LIN {X 52, Y 256, Z 47} c_vel
LIN {X 42, Y 261, Z 47} c_vel
LIN {X 30, Y 267, Z 47} c_vel
LIN {X 16, Y 273, Z 47} c_vel
LIN {X 0, Y 278, Z 47} c_vel
LIN {X 14, Y 327, Z 47} c_vel
LIN {X 28, Y 322, Z 47} c_vel
LIN {X 43, Y 317, Z 47} c_vel
LIN {X 57, Y 311, Z 47} c_vel
LIN {X 70, Y 304, Z 47} c_vel
LIN {X 81, Y 298, Z 47} c_vel
LIN {X 90, Y 291, Z 47} c_vel
LIN {X 99, Y 284, Z 47} c_vel
LIN {X 106, Y 277, Z 47} c_vel
LIN {X 113, Y 269, Z 47} c_vel
LIN {X 118, Y 261, Z 47} c_vel
LIN {X 123, Y 253, Z 47} c_vel
LIN {X 127, Y 244, Z 47} c_vel
LIN {X 130, Y 235, Z 47} c_vel
LIN {X 131, Y 226, Z 47} c_vel
LIN {X 133, Y 217, Z 47} c_vel
LIN {X 133, Y 207, Z 47} c_vel
LIN {X 133, Y 197, Z 47} c_vel
LIN {X 131, Y 186, Z 47} c_vel
LIN {X 129, Y 173, Z 47} c_vel
LIN {X 126, Y 160, Z 47} c_vel
LIN {X 120, Y 138, Z 47} c_vel
LIN {X 115, Y 118, Z 47} c_vel
LIN {X 112, Y 106, Z 47} c_vel
LIN {X 111, Y 96, Z 47} c_vel
LIN {X 110, Y 88, Z 47} c_vel
LIN {X 110, Y 81, Z 47} c_vel
LIN {X 111, Y 74, Z 47} c_vel
LIN {X 113, Y 69, Z 47} c_vel
LIN {X 116, Y 63, Z 47} c_vel
LIN {X 119, Y 58, Z 47} c_vel
LIN {X 124, Y 53, Z 47} c_vel
LIN {X 130, Y 48, Z 47} c_vel
LIN {X 138, Y 43, Z 47} c_vel
LIN {X 111, Y 0, Z 47} c_vel
$OUT[4] = FALSE
WAIT SEC 10.0
LIN {X 111, Y 0, Z 48} c_vel
$OUT[4] = TRUE
LIN {X 111, Y 0, Z 48} c_vel
LIN {X 106, Y 3, Z 48} c_vel
LIN {X 97, Y 9, Z 48} c_vel
LIN {X 89, Y 16, Z 48} c_vel
LIN {X 83, Y 23, Z 48} c_vel
LIN {X 77, Y 31, Z 48} c_vel
LIN {X 71, Y 39, Z 48} c_vel
LIN {X 67, Y 47, Z 48} c_vel
LIN {X 64, Y 56, Z 48} c_vel
LIN {X 62, Y 64, Z 48} c_vel
LIN {X 60, Y 73, Z 48} c_vel
LIN {X 59, Y 82, Z 48} c_vel
LIN {X 59, Y 92, Z 48} c_vel
LIN {X 60, Y 103, Z 48} c_vel
LIN {X 62, Y 114, Z 48} c_vel
LIN {X 65, Y 127, Z 48} c_vel
LIN {X 69, Y 144, Z 48} c_vel
LIN {X 74, Y 163, Z 48} c_vel
LIN {X 79, Y 180, Z 48} c_vel
LIN {X 81, Y 191, Z 48} c_vel
LIN {X 82, Y 201, Z 48} c_vel
LIN {X 82, Y 209, Z 48} c_vel
LIN {X 82, Y 217, Z 48} c_vel
LIN {X 80, Y 223, Z 48} c_vel
LIN {X 78, Y 229, Z 48} c_vel
LIN {X 75, Y 234, Z 48} c_vel
LIN {X 71, Y 240, Z 48} c_vel
LIN {X 66, Y 245, Z 48} c_vel
LIN {X 60, Y 250, Z 48} c_vel
LIN {X 52, Y 256, Z 48} c_vel
LIN {X 42, Y 261, Z 48} c_vel
LIN {X 30, Y 267, Z 48} c_vel
LIN {X 16, Y 273, Z 48} c_vel
LIN {X 0, Y 278, Z 48} c_vel
LIN {X 14, Y 327, Z 48} c_vel
LIN {X 28, Y 322, Z 48} c_vel
LIN {X 43, Y 317, Z 48} c_vel
LIN {X 57, Y 311, Z 48} c_vel
LIN {X 70, Y 304, Z 48} c_vel
LIN {X 81, Y 298, Z 48} c_vel
LIN {X 90, Y 291, Z 48} c_vel
LIN {X 99, Y 284, Z 48} c_vel
LIN {X 106, Y 277, Z 48} c_vel
LIN {X 113, Y 269, Z 48} c_vel
LIN {X 118, Y 261, Z 48} c_vel
LIN {X 123, Y 253, Z 48} c_vel
LIN {X 127, Y 244, Z 48} c_vel
LIN {X 130, Y 235, Z 48} c_vel
LIN {X 131, Y 226, Z 48} c_vel
LIN {X 133, Y 217, Z 48} c_vel
LIN {X 133, Y 207, Z 48} c_vel
LIN {X 133, Y 197, Z 48} c_vel
LIN {X 131, Y 186, Z 48} c_vel
LIN {X 129, Y 173, Z 48} c_vel
LIN {X 126, Y 160, Z 48} c_vel
LIN {X 120, Y 138, Z 48} c_vel
LIN {X 115, Y 118, Z 48} c_vel
LIN {X 112, Y 106, Z 48} c_vel
LIN {X 111, Y 96, Z 48} c_vel
LIN {X 110, Y 88, Z 48} c_vel
LIN {X 110, Y 81, Z 48} c_vel
LIN {X 111, Y 74, Z 48} c_vel
LIN {X 113, Y 69, Z 48} c_vel
LIN {X 116, Y 63, Z 48} c_vel
LIN {X 119, Y 58, Z 48} c_vel
LIN {X 124, Y 53, Z 48} c_vel
LIN {X 130, Y 48, Z 48} c_vel
LIN {X 138, Y 43, Z 48} c_vel
LIN {X 111, Y 0, Z 48} c_vel
$OUT[4] = FALSE
WAIT SEC 10.0
LIN {X 111, Y 0, Z 49} c_vel
$OUT[4] = TRUE
LIN {X 111, Y 0, Z 49} c_vel
LIN {X 106, Y 3, Z 49} c_vel
LIN {X 97, Y 9, Z 49} c_vel
LIN {X 89, Y 16, Z 49} c_vel
LIN {X 83, Y 23, Z 49} c_vel
LIN {X 77, Y 31, Z 49} c_vel
LIN {X 71, Y 39, Z 49} c_vel
LIN {X 67, Y 47, Z 49} c_vel
LIN {X 64, Y 56, Z 49} c_vel
LIN {X 62, Y 64, Z 49} c_vel
LIN {X 60, Y 73, Z 49} c_vel
LIN {X 59, Y 82, Z 49} c_vel
LIN {X 59, Y 92, Z 49} c_vel
LIN {X 60, Y 103, Z 49} c_vel
LIN {X 62, Y 114, Z 49} c_vel
LIN {X 65, Y 127, Z 49} c_vel
LIN {X 69, Y 144, Z 49} c_vel
LIN {X 74, Y 163, Z 49} c_vel
LIN {X 79, Y 180, Z 49} c_vel
LIN {X 81, Y 191, Z 49} c_vel
LIN {X 82, Y 201, Z 49} c_vel
LIN {X 82, Y 209, Z 49} c_vel
LIN {X 82, Y 217, Z 49} c_vel
LIN {X 80, Y 223, Z 49} c_vel
LIN {X 78, Y 229, Z 49} c_vel
LIN {X 75, Y 234, Z 49} c_vel
LIN {X 71, Y 240, Z 49} c_vel
LIN {X 66, Y 245, Z 49} c_vel
LIN {X 60, Y 250, Z 49} c_vel
LIN {X 52, Y 256, Z 49} c_vel
LIN {X 42, Y 261, Z 49} c_vel
LIN {X 30, Y 267, Z 49} c_vel
LIN {X 16, Y 273, Z 49} c_vel
LIN {X 0, Y 278, Z 49} c_vel
LIN {X 14, Y 327, Z 49} c_vel
LIN {X 28, Y 322, Z 49} c_vel
LIN {X 43, Y 317, Z 49} c_vel
LIN {X 57, Y 311, Z 49} c_vel
LIN {X 70, Y 304, Z 49} c_vel
LIN {X 81, Y 298, Z 49} c_vel
LIN {X 90, Y 291, Z 49} c_vel
LIN {X 99, Y 284, Z 49} c_vel
LIN {X 106, Y 277, Z 49} c_vel
LIN {X 113, Y 269, Z 49} c_vel
LIN {X 118, Y 261, Z 49} c_vel
LIN {X 123, Y 253, Z 49} c_vel
LIN {X 127, Y 244, Z 49} c_vel
LIN {X 130, Y 235, Z 49} c_vel
LIN {X 131, Y 226, Z 49} c_vel
LIN {X 133, Y 217, Z 49} c_vel
LIN {X 133, Y 207, Z 49} c_vel
LIN {X 133, Y 197, Z 49} c_vel
LIN {X 131, Y 186, Z 49} c_vel
LIN {X 129, Y 173, Z 49} c_vel
LIN {X 126, Y 160, Z 49} c_vel
LIN {X 120, Y 138, Z 49} c_vel
LIN {X 115, Y 118, Z 49} c_vel
LIN {X 112, Y 106, Z 49} c_vel
LIN {X 111, Y 96, Z 49} c_vel
LIN {X 110, Y 88, Z 49} c_vel
LIN {X 110, Y 81, Z 49} c_vel
LIN {X 111, Y 74, Z 49} c_vel
LIN {X 113, Y 69, Z 49} c_vel
LIN {X 116, Y 63, Z 49} c_vel
LIN {X 119, Y 58, Z 49} c_vel
LIN {X 124, Y 53, Z 49} c_vel
LIN {X 130, Y 48, Z 49} c_vel
LIN {X 138, Y 43, Z 49} c_vel
LIN {X 111, Y 0, Z 49} c_vel
$OUT[4] = FALSE
WAIT SEC 10.0
LIN {X 111, Y 0, Z 50} c_vel
$OUT[4] = TRUE
LIN {X 111, Y 0, Z 50} c_vel
LIN {X 106, Y 3, Z 50} c_vel
LIN {X 97, Y 9, Z 50} c_vel
LIN {X 89, Y 16, Z 50} c_vel
LIN {X 83, Y 23, Z 50} c_vel
LIN {X 77, Y 31, Z 50} c_vel
LIN {X 71, Y 39, Z 50} c_vel
LIN {X 67, Y 47, Z 50} c_vel
LIN {X 64, Y 56, Z 50} c_vel
LIN {X 62, Y 64, Z 50} c_vel
LIN {X 60, Y 73, Z 50} c_vel
LIN {X 59, Y 82, Z 50} c_vel
LIN {X 59, Y 92, Z 50} c_vel
LIN {X 60, Y 103, Z 50} c_vel
LIN {X 62, Y 114, Z 50} c_vel
LIN {X 65, Y 127, Z 50} c_vel
LIN {X 69, Y 144, Z 50} c_vel
LIN {X 74, Y 163, Z 50} c_vel
LIN {X 79, Y 180, Z 50} c_vel
LIN {X 81, Y 191, Z 50} c_vel
LIN {X 82, Y 201, Z 50} c_vel
LIN {X 82, Y 209, Z 50} c_vel
LIN {X 82, Y 217, Z 50} c_vel
LIN {X 80, Y 223, Z 50} c_vel
LIN {X 78, Y 229, Z 50} c_vel
LIN {X 75, Y 234, Z 50} c_vel
LIN {X 71, Y 240, Z 50} c_vel
LIN {X 66, Y 245, Z 50} c_vel
LIN {X 60, Y 250, Z 50} c_vel
LIN {X 52, Y 256, Z 50} c_vel
LIN {X 42, Y 261, Z 50} c_vel
LIN {X 30, Y 267, Z 50} c_vel
LIN {X 16, Y 273, Z 50} c_vel
LIN {X 0, Y 278, Z 50} c_vel
LIN {X 14, Y 327, Z 50} c_vel
LIN {X 28, Y 322, Z 50} c_vel
LIN {X 43, Y 317, Z 50} c_vel
LIN {X 57, Y 311, Z 50} c_vel
LIN {X 70, Y 304, Z 50} c_vel
LIN {X 81, Y 298, Z 50} c_vel
LIN {X 90, Y 291, Z 50} c_vel
LIN {X 99, Y 284, Z 50} c_vel
LIN {X 106, Y 277, Z 50} c_vel
LIN {X 113, Y 269, Z 50} c_vel
LIN {X 118, Y 261, Z 50} c_vel
LIN {X 123, Y 253, Z 50} c_vel
LIN {X 127, Y 244, Z 50} c_vel
LIN {X 130, Y 235, Z 50} c_vel
LIN {X 131, Y 226, Z 50} c_vel
LIN {X 133, Y 217, Z 50} c_vel
LIN {X 133, Y 207, Z 50} c_vel
LIN {X 133, Y 197, Z 50} c_vel
LIN {X 131, Y 186, Z 50} c_vel
LIN {X 129, Y 173, Z 50} c_vel
LIN {X 126, Y 160, Z 50} c_vel
LIN {X 120, Y 138, Z 50} c_vel
LIN {X 115, Y 118, Z 50} c_vel
LIN {X 112, Y 106, Z 50} c_vel
LIN {X 111, Y 96, Z 50} c_vel
LIN {X 110, Y 88, Z 50} c_vel
LIN {X 110, Y 81, Z 50} c_vel
LIN {X 111, Y 74, Z 50} c_vel
LIN {X 113, Y 69, Z 50} c_vel
LIN {X 116, Y 63, Z 50} c_vel
LIN {X 119, Y 58, Z 50} c_vel
LIN {X 124, Y 53, Z 50} c_vel
LIN {X 130, Y 48, Z 50} c_vel
LIN {X 138, Y 43, Z 50} c_vel
LIN {X 111, Y 0, Z 50} c_vel
$OUT[4] = FALSE
WAIT SEC 10.0
LIN {X 111, Y 0, Z 51} c_vel
$OUT[4] = TRUE
LIN {X 111, Y 0, Z 51} c_vel
LIN {X 106, Y 3, Z 51} c_vel
LIN {X 97, Y 9, Z 51} c_vel
LIN {X 89, Y 16, Z 51} c_vel
LIN {X 83, Y 23, Z 51} c_vel
LIN {X 77, Y 31, Z 51} c_vel
LIN {X 71, Y 39, Z 51} c_vel
LIN {X 67, Y 47, Z 51} c_vel
LIN {X 64, Y 56, Z 51} c_vel
LIN {X 62, Y 64, Z 51} c_vel
LIN {X 60, Y 73, Z 51} c_vel
LIN {X 59, Y 82, Z 51} c_vel
LIN {X 59, Y 92, Z 51} c_vel
LIN {X 60, Y 103, Z 51} c_vel
LIN {X 62, Y 114, Z 51} c_vel
LIN {X 65, Y 127, Z 51} c_vel
LIN {X 69, Y 144, Z 51} c_vel
LIN {X 74, Y 163, Z 51} c_vel
LIN {X 79, Y 180, Z 51} c_vel
LIN {X 81, Y 191, Z 51} c_vel
LIN {X 82, Y 201, Z 51} c_vel
LIN {X 82, Y 209, Z 51} c_vel
LIN {X 82, Y 217, Z 51} c_vel
LIN {X 80, Y 223, Z 51} c_vel
LIN {X 78, Y 229, Z 51} c_vel
LIN {X 75, Y 234, Z 51} c_vel
LIN {X 71, Y 240, Z 51} c_vel
LIN {X 66, Y 245, Z 51} c_vel
LIN {X 60, Y 250, Z 51} c_vel
LIN {X 52, Y 256, Z 51} c_vel
LIN {X 42, Y 261, Z 51} c_vel
LIN {X 30, Y 267, Z 51} c_vel
LIN {X 16, Y 273, Z 51} c_vel
LIN {X 0, Y 278, Z 51} c_vel
LIN {X 14, Y 327, Z 51} c_vel
LIN {X 28, Y 322, Z 51} c_vel
LIN {X 43, Y 317, Z 51} c_vel
LIN {X 57, Y 311, Z 51} c_vel
LIN {X 70, Y 304, Z 51} c_vel
LIN {X 81, Y 298, Z 51} c_vel
LIN {X 90, Y 291, Z 51} c_vel
LIN {X 99, Y 284, Z 51} c_vel
LIN {X 106, Y 277, Z 51} c_vel
LIN {X 113, Y 269, Z 51} c_vel
LIN {X 118, Y 261, Z 51} c_vel
LIN {X 123, Y 253, Z 51} c_vel
LIN {X 127, Y 244, Z 51} c_vel
LIN {X 130, Y 235, Z 51} c_vel
LIN {X 131, Y 226, Z 51} c_vel
LIN {X 133, Y 217, Z 51} c_vel
LIN {X 133, Y 207, Z 51} c_vel
LIN {X 133, Y 197, Z 51} c_vel
LIN {X 131, Y 186, Z 51} c_vel
LIN {X 129, Y 173, Z 51} c_vel
LIN {X 126, Y 160, Z 51} c_vel
LIN {X 120, Y 138, Z 51} c_vel
LIN {X 115, Y 118, Z 51} c_vel
LIN {X 112, Y 106, Z 51} c_vel
LIN {X 111, Y 96, Z 51} c_vel
LIN {X 110, Y 88, Z 51} c_vel
LIN {X 110, Y 81, Z 51} c_vel
LIN {X 111, Y 74, Z 51} c_vel
LIN {X 113, Y 69, Z 51} c_vel
LIN {X 116, Y 63, Z 51} c_vel
LIN {X 119, Y 58, Z 51} c_vel
LIN {X 124, Y 53, Z 51} c_vel
LIN {X 130, Y 48, Z 51} c_vel
LIN {X 138, Y 43, Z 51} c_vel
LIN {X 111, Y 0, Z 51} c_vel
$OUT[4] = FALSE
WAIT SEC 10.0
LIN {X 111, Y 0, Z 52} c_vel
$OUT[4] = TRUE
LIN {X 111, Y 0, Z 52} c_vel
LIN {X 106, Y 3, Z 52} c_vel
LIN {X 97, Y 9, Z 52} c_vel
LIN {X 89, Y 16, Z 52} c_vel
LIN {X 83, Y 23, Z 52} c_vel
LIN {X 77, Y 31, Z 52} c_vel
LIN {X 71, Y 39, Z 52} c_vel
LIN {X 67, Y 47, Z 52} c_vel
LIN {X 64, Y 56, Z 52} c_vel
LIN {X 62, Y 64, Z 52} c_vel
LIN {X 60, Y 73, Z 52} c_vel
LIN {X 59, Y 82, Z 52} c_vel
LIN {X 59, Y 92, Z 52} c_vel
LIN {X 60, Y 103, Z 52} c_vel
LIN {X 62, Y 114, Z 52} c_vel
LIN {X 65, Y 127, Z 52} c_vel
LIN {X 69, Y 144, Z 52} c_vel
LIN {X 74, Y 163, Z 52} c_vel
LIN {X 79, Y 180, Z 52} c_vel
LIN {X 81, Y 191, Z 52} c_vel
LIN {X 82, Y 201, Z 52} c_vel
LIN {X 82, Y 209, Z 52} c_vel
LIN {X 82, Y 217, Z 52} c_vel
LIN {X 80, Y 223, Z 52} c_vel
LIN {X 78, Y 229, Z 52} c_vel
LIN {X 75, Y 234, Z 52} c_vel
LIN {X 71, Y 240, Z 52} c_vel
LIN {X 66, Y 245, Z 52} c_vel
LIN {X 60, Y 250, Z 52} c_vel
LIN {X 52, Y 256, Z 52} c_vel
LIN {X 42, Y 261, Z 52} c_vel
LIN {X 30, Y 267, Z 52} c_vel
LIN {X 16, Y 273, Z 52} c_vel
LIN {X 0, Y 278, Z 52} c_vel
LIN {X 14, Y 327, Z 52} c_vel
LIN {X 28, Y 322, Z 52} c_vel
LIN {X 43, Y 317, Z 52} c_vel
LIN {X 57, Y 311, Z 52} c_vel
LIN {X 70, Y 304, Z 52} c_vel
LIN {X 81, Y 298, Z 52} c_vel
LIN {X 90, Y 291, Z 52} c_vel
LIN {X 99, Y 284, Z 52} c_vel
LIN {X 106, Y 277, Z 52} c_vel
LIN {X 113, Y 269, Z 52} c_vel
LIN {X 118, Y 261, Z 52} c_vel
LIN {X 123, Y 253, Z 52} c_vel
LIN {X 127, Y 244, Z 52} c_vel
LIN {X 130, Y 235, Z 52} c_vel
LIN {X 131, Y 226, Z 52} c_vel
LIN {X 133, Y 217, Z 52} c_vel
LIN {X 133, Y 207, Z 52} c_vel
LIN {X 133, Y 197, Z 52} c_vel
LIN {X 131, Y 186, Z 52} c_vel
LIN {X 129, Y 173, Z 52} c_vel
LIN {X 126, Y 160, Z 52} c_vel
LIN {X 120, Y 138, Z 52} c_vel
LIN {X 115, Y 118, Z 52} c_vel
LIN {X 112, Y 106, Z 52} c_vel
LIN {X 111, Y 96, Z 52} c_vel
LIN {X 110, Y 88, Z 52} c_vel
LIN {X 110, Y 81, Z 52} c_vel
LIN {X 111, Y 74, Z 52} c_vel
LIN {X 113, Y 69, Z 52} c_vel
LIN {X 116, Y 63, Z 52} c_vel
LIN {X 119, Y 58, Z 52} c_vel
LIN {X 124, Y 53, Z 52} c_vel
LIN {X 130, Y 48, Z 52} c_vel
LIN {X 138, Y 43, Z 52} c_vel
LIN {X 111, Y 0, Z 52} c_vel
$OUT[4] = FALSE
WAIT SEC 10.0
LIN {X 111, Y 0, Z 53} c_vel
$OUT[4] = TRUE
LIN {X 111, Y 0, Z 53} c_vel
LIN {X 106, Y 3, Z 53} c_vel
LIN {X 97, Y 9, Z 53} c_vel
LIN {X 89, Y 16, Z 53} c_vel
LIN {X 83, Y 23, Z 53} c_vel
LIN {X 77, Y 31, Z 53} c_vel
LIN {X 71, Y 39, Z 53} c_vel
LIN {X 67, Y 47, Z 53} c_vel
LIN {X 64, Y 56, Z 53} c_vel
LIN {X 62, Y 64, Z 53} c_vel
LIN {X 60, Y 73, Z 53} c_vel
LIN {X 59, Y 82, Z 53} c_vel
LIN {X 59, Y 92, Z 53} c_vel
LIN {X 60, Y 103, Z 53} c_vel
LIN {X 62, Y 114, Z 53} c_vel
LIN {X 65, Y 127, Z 53} c_vel
LIN {X 69, Y 144, Z 53} c_vel
LIN {X 74, Y 163, Z 53} c_vel
LIN {X 79, Y 180, Z 53} c_vel
LIN {X 81, Y 191, Z 53} c_vel
LIN {X 82, Y 201, Z 53} c_vel
LIN {X 82, Y 209, Z 53} c_vel
LIN {X 82, Y 217, Z 53} c_vel
LIN {X 80, Y 223, Z 53} c_vel
LIN {X 78, Y 229, Z 53} c_vel
LIN {X 75, Y 234, Z 53} c_vel
LIN {X 71, Y 240, Z 53} c_vel
LIN {X 66, Y 245, Z 53} c_vel
LIN {X 60, Y 250, Z 53} c_vel
LIN {X 52, Y 256, Z 53} c_vel
LIN {X 42, Y 261, Z 53} c_vel
LIN {X 30, Y 267, Z 53} c_vel
LIN {X 16, Y 273, Z 53} c_vel
LIN {X 0, Y 278, Z 53} c_vel
LIN {X 14, Y 327, Z 53} c_vel
LIN {X 28, Y 322, Z 53} c_vel
LIN {X 43, Y 317, Z 53} c_vel
LIN {X 57, Y 311, Z 53} c_vel
LIN {X 70, Y 304, Z 53} c_vel
LIN {X 81, Y 298, Z 53} c_vel
LIN {X 90, Y 291, Z 53} c_vel
LIN {X 99, Y 284, Z 53} c_vel
LIN {X 106, Y 277, Z 53} c_vel
LIN {X 113, Y 269, Z 53} c_vel
LIN {X 118, Y 261, Z 53} c_vel
LIN {X 123, Y 253, Z 53} c_vel
LIN {X 127, Y 244, Z 53} c_vel
LIN {X 130, Y 235, Z 53} c_vel
LIN {X 131, Y 226, Z 53} c_vel
LIN {X 133, Y 217, Z 53} c_vel
LIN {X 133, Y 207, Z 53} c_vel
LIN {X 133, Y 197, Z 53} c_vel
LIN {X 131, Y 186, Z 53} c_vel
LIN {X 129, Y 173, Z 53} c_vel
LIN {X 126, Y 160, Z 53} c_vel
LIN {X 120, Y 138, Z 53} c_vel
LIN {X 115, Y 118, Z 53} c_vel
LIN {X 112, Y 106, Z 53} c_vel
LIN {X 111, Y 96, Z 53} c_vel
LIN {X 110, Y 88, Z 53} c_vel
LIN {X 110, Y 81, Z 53} c_vel
LIN {X 111, Y 74, Z 53} c_vel
LIN {X 113, Y 69, Z 53} c_vel
LIN {X 116, Y 63, Z 53} c_vel
LIN {X 119, Y 58, Z 53} c_vel
LIN {X 124, Y 53, Z 53} c_vel
LIN {X 130, Y 48, Z 53} c_vel
LIN {X 138, Y 43, Z 53} c_vel
LIN {X 111, Y 0, Z 53} c_vel
$OUT[4] = FALSE
WAIT SEC 10.0
LIN {X 111, Y 0, Z 54} c_vel
$OUT[4] = TRUE
LIN {X 111, Y 0, Z 54} c_vel
LIN {X 106, Y 3, Z 54} c_vel
LIN {X 97, Y 9, Z 54} c_vel
LIN {X 89, Y 16, Z 54} c_vel
LIN {X 83, Y 23, Z 54} c_vel
LIN {X 77, Y 31, Z 54} c_vel
LIN {X 71, Y 39, Z 54} c_vel
LIN {X 67, Y 47, Z 54} c_vel
LIN {X 64, Y 56, Z 54} c_vel
LIN {X 62, Y 64, Z 54} c_vel
LIN {X 60, Y 73, Z 54} c_vel
LIN {X 59, Y 82, Z 54} c_vel
LIN {X 59, Y 92, Z 54} c_vel
LIN {X 60, Y 103, Z 54} c_vel
LIN {X 62, Y 114, Z 54} c_vel
LIN {X 65, Y 127, Z 54} c_vel
LIN {X 69, Y 144, Z 54} c_vel
LIN {X 74, Y 163, Z 54} c_vel
LIN {X 79, Y 180, Z 54} c_vel
LIN {X 81, Y 191, Z 54} c_vel
LIN {X 82, Y 201, Z 54} c_vel
LIN {X 82, Y 209, Z 54} c_vel
LIN {X 82, Y 217, Z 54} c_vel
LIN {X 80, Y 223, Z 54} c_vel
LIN {X 78, Y 229, Z 54} c_vel
LIN {X 75, Y 234, Z 54} c_vel
LIN {X 71, Y 240, Z 54} c_vel
LIN {X 66, Y 245, Z 54} c_vel
LIN {X 60, Y 250, Z 54} c_vel
LIN {X 52, Y 256, Z 54} c_vel
LIN {X 42, Y 261, Z 54} c_vel
LIN {X 30, Y 267, Z 54} c_vel
LIN {X 16, Y 273, Z 54} c_vel
LIN {X 0, Y 278, Z 54} c_vel
LIN {X 14, Y 327, Z 54} c_vel
LIN {X 28, Y 322, Z 54} c_vel
LIN {X 43, Y 317, Z 54} c_vel
LIN {X 57, Y 311, Z 54} c_vel
LIN {X 70, Y 304, Z 54} c_vel
LIN {X 81, Y 298, Z 54} c_vel
LIN {X 90, Y 291, Z 54} c_vel
LIN {X 99, Y 284, Z 54} c_vel
LIN {X 106, Y 277, Z 54} c_vel
LIN {X 113, Y 269, Z 54} c_vel
LIN {X 118, Y 261, Z 54} c_vel
LIN {X 123, Y 253, Z 54} c_vel
LIN {X 127, Y 244, Z 54} c_vel
LIN {X 130, Y 235, Z 54} c_vel
LIN {X 131, Y 226, Z 54} c_vel
LIN {X 133, Y 217, Z 54} c_vel
LIN {X 133, Y 207, Z 54} c_vel
LIN {X 133, Y 197, Z 54} c_vel
LIN {X 131, Y 186, Z 54} c_vel
LIN {X 129, Y 173, Z 54} c_vel
LIN {X 126, Y 160, Z 54} c_vel
LIN {X 120, Y 138, Z 54} c_vel
LIN {X 115, Y 118, Z 54} c_vel
LIN {X 112, Y 106, Z 54} c_vel
LIN {X 111, Y 96, Z 54} c_vel
LIN {X 110, Y 88, Z 54} c_vel
LIN {X 110, Y 81, Z 54} c_vel
LIN {X 111, Y 74, Z 54} c_vel
LIN {X 113, Y 69, Z 54} c_vel
LIN {X 116, Y 63, Z 54} c_vel
LIN {X 119, Y 58, Z 54} c_vel
LIN {X 124, Y 53, Z 54} c_vel
LIN {X 130, Y 48, Z 54} c_vel
LIN {X 138, Y 43, Z 54} c_vel
LIN {X 111, Y 0, Z 54} c_vel
$OUT[4] = FALSE
WAIT SEC 10.0
LIN {X 111, Y 0, Z 55} c_vel
$OUT[4] = TRUE
LIN {X 111, Y 0, Z 55} c_vel
LIN {X 106, Y 3, Z 55} c_vel
LIN {X 97, Y 9, Z 55} c_vel
LIN {X 89, Y 16, Z 55} c_vel
LIN {X 83, Y 23, Z 55} c_vel
LIN {X 77, Y 31, Z 55} c_vel
LIN {X 71, Y 39, Z 55} c_vel
LIN {X 67, Y 47, Z 55} c_vel
LIN {X 64, Y 56, Z 55} c_vel
LIN {X 62, Y 64, Z 55} c_vel
LIN {X 60, Y 73, Z 55} c_vel
LIN {X 59, Y 82, Z 55} c_vel
LIN {X 59, Y 92, Z 55} c_vel
LIN {X 60, Y 103, Z 55} c_vel
LIN {X 62, Y 114, Z 55} c_vel
LIN {X 65, Y 127, Z 55} c_vel
LIN {X 69, Y 144, Z 55} c_vel
LIN {X 74, Y 163, Z 55} c_vel
LIN {X 79, Y 180, Z 55} c_vel
LIN {X 81, Y 191, Z 55} c_vel
LIN {X 82, Y 201, Z 55} c_vel
LIN {X 82, Y 209, Z 55} c_vel
LIN {X 82, Y 217, Z 55} c_vel
LIN {X 80, Y 223, Z 55} c_vel
LIN {X 78, Y 229, Z 55} c_vel
LIN {X 75, Y 234, Z 55} c_vel
LIN {X 71, Y 240, Z 55} c_vel
LIN {X 66, Y 245, Z 55} c_vel
LIN {X 60, Y 250, Z 55} c_vel
LIN {X 52, Y 256, Z 55} c_vel
LIN {X 42, Y 261, Z 55} c_vel
LIN {X 30, Y 267, Z 55} c_vel
LIN {X 16, Y 273, Z 55} c_vel
LIN {X 0, Y 278, Z 55} c_vel
LIN {X 14, Y 327, Z 55} c_vel
LIN {X 28, Y 322, Z 55} c_vel
LIN {X 43, Y 317, Z 55} c_vel
LIN {X 57, Y 311, Z 55} c_vel
LIN {X 70, Y 304, Z 55} c_vel
LIN {X 81, Y 298, Z 55} c_vel
LIN {X 90, Y 291, Z 55} c_vel
LIN {X 99, Y 284, Z 55} c_vel
LIN {X 106, Y 277, Z 55} c_vel
LIN {X 113, Y 269, Z 55} c_vel
LIN {X 118, Y 261, Z 55} c_vel
LIN {X 123, Y 253, Z 55} c_vel
LIN {X 127, Y 244, Z 55} c_vel
LIN {X 130, Y 235, Z 55} c_vel
LIN {X 131, Y 226, Z 55} c_vel
LIN {X 133, Y 217, Z 55} c_vel
LIN {X 133, Y 207, Z 55} c_vel
LIN {X 133, Y 197, Z 55} c_vel
LIN {X 131, Y 186, Z 55} c_vel
LIN {X 129, Y 173, Z 55} c_vel
LIN {X 126, Y 160, Z 55} c_vel
LIN {X 120, Y 138, Z 55} c_vel
LIN {X 115, Y 118, Z 55} c_vel
LIN {X 112, Y 106, Z 55} c_vel
LIN {X 111, Y 96, Z 55} c_vel
LIN {X 110, Y 88, Z 55} c_vel
LIN {X 110, Y 81, Z 55} c_vel
LIN {X 111, Y 74, Z 55} c_vel
LIN {X 113, Y 69, Z 55} c_vel
LIN {X 116, Y 63, Z 55} c_vel
LIN {X 119, Y 58, Z 55} c_vel
LIN {X 124, Y 53, Z 55} c_vel
LIN {X 130, Y 48, Z 55} c_vel
LIN {X 138, Y 43, Z 55} c_vel
LIN {X 111, Y 0, Z 55} c_vel
$OUT[4] = FALSE
WAIT SEC 10.0
LIN {X 111, Y 0, Z 56} c_vel
$OUT[4] = TRUE
LIN {X 111, Y 0, Z 56} c_vel
LIN {X 106, Y 3, Z 56} c_vel
LIN {X 97, Y 9, Z 56} c_vel
LIN {X 89, Y 16, Z 56} c_vel
LIN {X 83, Y 23, Z 56} c_vel
LIN {X 77, Y 31, Z 56} c_vel
LIN {X 71, Y 39, Z 56} c_vel
LIN {X 67, Y 47, Z 56} c_vel
LIN {X 64, Y 56, Z 56} c_vel
LIN {X 62, Y 64, Z 56} c_vel
LIN {X 60, Y 73, Z 56} c_vel
LIN {X 59, Y 82, Z 56} c_vel
LIN {X 59, Y 92, Z 56} c_vel
LIN {X 60, Y 103, Z 56} c_vel
LIN {X 62, Y 114, Z 56} c_vel
LIN {X 65, Y 127, Z 56} c_vel
LIN {X 69, Y 144, Z 56} c_vel
LIN {X 74, Y 163, Z 56} c_vel
LIN {X 79, Y 180, Z 56} c_vel
LIN {X 81, Y 191, Z 56} c_vel
LIN {X 82, Y 201, Z 56} c_vel
LIN {X 82, Y 209, Z 56} c_vel
LIN {X 82, Y 217, Z 56} c_vel
LIN {X 80, Y 223, Z 56} c_vel
LIN {X 78, Y 229, Z 56} c_vel
LIN {X 75, Y 234, Z 56} c_vel
LIN {X 71, Y 240, Z 56} c_vel
LIN {X 66, Y 245, Z 56} c_vel
LIN {X 60, Y 250, Z 56} c_vel
LIN {X 52, Y 256, Z 56} c_vel
LIN {X 42, Y 261, Z 56} c_vel
LIN {X 30, Y 267, Z 56} c_vel
LIN {X 16, Y 273, Z 56} c_vel
LIN {X 0, Y 278, Z 56} c_vel
LIN {X 14, Y 327, Z 56} c_vel
LIN {X 28, Y 322, Z 56} c_vel
LIN {X 43, Y 317, Z 56} c_vel
LIN {X 57, Y 311, Z 56} c_vel
LIN {X 70, Y 304, Z 56} c_vel
LIN {X 81, Y 298, Z 56} c_vel
LIN {X 90, Y 291, Z 56} c_vel
LIN {X 99, Y 284, Z 56} c_vel
LIN {X 106, Y 277, Z 56} c_vel
LIN {X 113, Y 269, Z 56} c_vel
LIN {X 118, Y 261, Z 56} c_vel
LIN {X 123, Y 253, Z 56} c_vel
LIN {X 127, Y 244, Z 56} c_vel
LIN {X 130, Y 235, Z 56} c_vel
LIN {X 131, Y 226, Z 56} c_vel
LIN {X 133, Y 217, Z 56} c_vel
LIN {X 133, Y 207, Z 56} c_vel
LIN {X 133, Y 197, Z 56} c_vel
LIN {X 131, Y 186, Z 56} c_vel
LIN {X 129, Y 173, Z 56} c_vel
LIN {X 126, Y 160, Z 56} c_vel
LIN {X 120, Y 138, Z 56} c_vel
LIN {X 115, Y 118, Z 56} c_vel
LIN {X 112, Y 106, Z 56} c_vel
LIN {X 111, Y 96, Z 56} c_vel
LIN {X 110, Y 88, Z 56} c_vel
LIN {X 110, Y 81, Z 56} c_vel
LIN {X 111, Y 74, Z 56} c_vel
LIN {X 113, Y 69, Z 56} c_vel
LIN {X 116, Y 63, Z 56} c_vel
LIN {X 119, Y 58, Z 56} c_vel
LIN {X 124, Y 53, Z 56} c_vel
LIN {X 130, Y 48, Z 56} c_vel
LIN {X 138, Y 43, Z 56} c_vel
LIN {X 111, Y 0, Z 56} c_vel
$OUT[4] = FALSE
WAIT SEC 10.0
LIN {X 111, Y 0, Z 57} c_vel
$OUT[4] = TRUE
LIN {X 111, Y 0, Z 57} c_vel
LIN {X 106, Y 3, Z 57} c_vel
LIN {X 97, Y 9, Z 57} c_vel
LIN {X 89, Y 16, Z 57} c_vel
LIN {X 83, Y 23, Z 57} c_vel
LIN {X 77, Y 31, Z 57} c_vel
LIN {X 71, Y 39, Z 57} c_vel
LIN {X 67, Y 47, Z 57} c_vel
LIN {X 64, Y 56, Z 57} c_vel
LIN {X 62, Y 64, Z 57} c_vel
LIN {X 60, Y 73, Z 57} c_vel
LIN {X 59, Y 82, Z 57} c_vel
LIN {X 59, Y 92, Z 57} c_vel
LIN {X 60, Y 103, Z 57} c_vel
LIN {X 62, Y 114, Z 57} c_vel
LIN {X 65, Y 127, Z 57} c_vel
LIN {X 69, Y 144, Z 57} c_vel
LIN {X 74, Y 163, Z 57} c_vel
LIN {X 79, Y 180, Z 57} c_vel
LIN {X 81, Y 191, Z 57} c_vel
LIN {X 82, Y 201, Z 57} c_vel
LIN {X 82, Y 209, Z 57} c_vel
LIN {X 82, Y 217, Z 57} c_vel
LIN {X 80, Y 223, Z 57} c_vel
LIN {X 78, Y 229, Z 57} c_vel
LIN {X 75, Y 234, Z 57} c_vel
LIN {X 71, Y 240, Z 57} c_vel
LIN {X 66, Y 245, Z 57} c_vel
LIN {X 60, Y 250, Z 57} c_vel
LIN {X 52, Y 256, Z 57} c_vel
LIN {X 42, Y 261, Z 57} c_vel
LIN {X 30, Y 267, Z 57} c_vel
LIN {X 16, Y 273, Z 57} c_vel
LIN {X 0, Y 278, Z 57} c_vel
LIN {X 14, Y 327, Z 57} c_vel
LIN {X 28, Y 322, Z 57} c_vel
LIN {X 43, Y 317, Z 57} c_vel
LIN {X 57, Y 311, Z 57} c_vel
LIN {X 70, Y 304, Z 57} c_vel
LIN {X 81, Y 298, Z 57} c_vel
LIN {X 90, Y 291, Z 57} c_vel
LIN {X 99, Y 284, Z 57} c_vel
LIN {X 106, Y 277, Z 57} c_vel
LIN {X 113, Y 269, Z 57} c_vel
LIN {X 118, Y 261, Z 57} c_vel
LIN {X 123, Y 253, Z 57} c_vel
LIN {X 127, Y 244, Z 57} c_vel
LIN {X 130, Y 235, Z 57} c_vel
LIN {X 131, Y 226, Z 57} c_vel
LIN {X 133, Y 217, Z 57} c_vel
LIN {X 133, Y 207, Z 57} c_vel
LIN {X 133, Y 197, Z 57} c_vel
LIN {X 131, Y 186, Z 57} c_vel
LIN {X 129, Y 173, Z 57} c_vel
LIN {X 126, Y 160, Z 57} c_vel
LIN {X 120, Y 138, Z 57} c_vel
LIN {X 115, Y 118, Z 57} c_vel
LIN {X 112, Y 106, Z 57} c_vel
LIN {X 111, Y 96, Z 57} c_vel
LIN {X 110, Y 88, Z 57} c_vel
LIN {X 110, Y 81, Z 57} c_vel
LIN {X 111, Y 74, Z 57} c_vel
LIN {X 113, Y 69, Z 57} c_vel
LIN {X 116, Y 63, Z 57} c_vel
LIN {X 119, Y 58, Z 57} c_vel
LIN {X 124, Y 53, Z 57} c_vel
LIN {X 130, Y 48, Z 57} c_vel
LIN {X 138, Y 43, Z 57} c_vel
LIN {X 111, Y 0, Z 57} c_vel
$OUT[4] = FALSE
WAIT SEC 10.0
LIN {X 111, Y 0, Z 58} c_vel
$OUT[4] = TRUE
LIN {X 111, Y 0, Z 58} c_vel
LIN {X 106, Y 3, Z 58} c_vel
LIN {X 97, Y 9, Z 58} c_vel
LIN {X 89, Y 16, Z 58} c_vel
LIN {X 83, Y 23, Z 58} c_vel
LIN {X 77, Y 31, Z 58} c_vel
LIN {X 71, Y 39, Z 58} c_vel
LIN {X 67, Y 47, Z 58} c_vel
LIN {X 64, Y 56, Z 58} c_vel
LIN {X 62, Y 64, Z 58} c_vel
LIN {X 60, Y 73, Z 58} c_vel
LIN {X 59, Y 82, Z 58} c_vel
LIN {X 59, Y 92, Z 58} c_vel
LIN {X 60, Y 103, Z 58} c_vel
LIN {X 62, Y 114, Z 58} c_vel
LIN {X 65, Y 127, Z 58} c_vel
LIN {X 69, Y 144, Z 58} c_vel
LIN {X 74, Y 163, Z 58} c_vel
LIN {X 79, Y 180, Z 58} c_vel
LIN {X 81, Y 191, Z 58} c_vel
LIN {X 82, Y 201, Z 58} c_vel
LIN {X 82, Y 209, Z 58} c_vel
LIN {X 82, Y 217, Z 58} c_vel
LIN {X 80, Y 223, Z 58} c_vel
LIN {X 78, Y 229, Z 58} c_vel
LIN {X 75, Y 234, Z 58} c_vel
LIN {X 71, Y 240, Z 58} c_vel
LIN {X 66, Y 245, Z 58} c_vel
LIN {X 60, Y 250, Z 58} c_vel
LIN {X 52, Y 256, Z 58} c_vel
LIN {X 42, Y 261, Z 58} c_vel
LIN {X 30, Y 267, Z 58} c_vel
LIN {X 16, Y 273, Z 58} c_vel
LIN {X 0, Y 278, Z 58} c_vel
LIN {X 14, Y 327, Z 58} c_vel
LIN {X 28, Y 322, Z 58} c_vel
LIN {X 43, Y 317, Z 58} c_vel
LIN {X 57, Y 311, Z 58} c_vel
LIN {X 70, Y 304, Z 58} c_vel
LIN {X 81, Y 298, Z 58} c_vel
LIN {X 90, Y 291, Z 58} c_vel
LIN {X 99, Y 284, Z 58} c_vel
LIN {X 106, Y 277, Z 58} c_vel
LIN {X 113, Y 269, Z 58} c_vel
LIN {X 118, Y 261, Z 58} c_vel
LIN {X 123, Y 253, Z 58} c_vel
LIN {X 127, Y 244, Z 58} c_vel
LIN {X 130, Y 235, Z 58} c_vel
LIN {X 131, Y 226, Z 58} c_vel
LIN {X 133, Y 217, Z 58} c_vel
LIN {X 133, Y 207, Z 58} c_vel
LIN {X 133, Y 197, Z 58} c_vel
LIN {X 131, Y 186, Z 58} c_vel
LIN {X 129, Y 173, Z 58} c_vel
LIN {X 126, Y 160, Z 58} c_vel
LIN {X 120, Y 138, Z 58} c_vel
LIN {X 115, Y 118, Z 58} c_vel
LIN {X 112, Y 106, Z 58} c_vel
LIN {X 111, Y 96, Z 58} c_vel
LIN {X 110, Y 88, Z 58} c_vel
LIN {X 110, Y 81, Z 58} c_vel
LIN {X 111, Y 74, Z 58} c_vel
LIN {X 113, Y 69, Z 58} c_vel
LIN {X 116, Y 63, Z 58} c_vel
LIN {X 119, Y 58, Z 58} c_vel
LIN {X 124, Y 53, Z 58} c_vel
LIN {X 130, Y 48, Z 58} c_vel
LIN {X 138, Y 43, Z 58} c_vel
LIN {X 111, Y 0, Z 58} c_vel
$OUT[4] = FALSE
WAIT SEC 10.0
LIN {X 111, Y 0, Z 59} c_vel
$OUT[4] = TRUE
LIN {X 111, Y 0, Z 59} c_vel
LIN {X 106, Y 3, Z 59} c_vel
LIN {X 97, Y 9, Z 59} c_vel
LIN {X 89, Y 16, Z 59} c_vel
LIN {X 83, Y 23, Z 59} c_vel
LIN {X 77, Y 31, Z 59} c_vel
LIN {X 71, Y 39, Z 59} c_vel
LIN {X 67, Y 47, Z 59} c_vel
LIN {X 64, Y 56, Z 59} c_vel
LIN {X 62, Y 64, Z 59} c_vel
LIN {X 60, Y 73, Z 59} c_vel
LIN {X 59, Y 82, Z 59} c_vel
LIN {X 59, Y 92, Z 59} c_vel
LIN {X 60, Y 103, Z 59} c_vel
LIN {X 62, Y 114, Z 59} c_vel
LIN {X 65, Y 127, Z 59} c_vel
LIN {X 69, Y 144, Z 59} c_vel
LIN {X 74, Y 163, Z 59} c_vel
LIN {X 79, Y 180, Z 59} c_vel
LIN {X 81, Y 191, Z 59} c_vel
LIN {X 82, Y 201, Z 59} c_vel
LIN {X 82, Y 209, Z 59} c_vel
LIN {X 82, Y 217, Z 59} c_vel
LIN {X 80, Y 223, Z 59} c_vel
LIN {X 78, Y 229, Z 59} c_vel
LIN {X 75, Y 234, Z 59} c_vel
LIN {X 71, Y 240, Z 59} c_vel
LIN {X 66, Y 245, Z 59} c_vel
LIN {X 60, Y 250, Z 59} c_vel
LIN {X 52, Y 256, Z 59} c_vel
LIN {X 42, Y 261, Z 59} c_vel
LIN {X 30, Y 267, Z 59} c_vel
LIN {X 16, Y 273, Z 59} c_vel
LIN {X 0, Y 278, Z 59} c_vel
LIN {X 14, Y 327, Z 59} c_vel
LIN {X 28, Y 322, Z 59} c_vel
LIN {X 43, Y 317, Z 59} c_vel
LIN {X 57, Y 311, Z 59} c_vel
LIN {X 70, Y 304, Z 59} c_vel
LIN {X 81, Y 298, Z 59} c_vel
LIN {X 90, Y 291, Z 59} c_vel
LIN {X 99, Y 284, Z 59} c_vel
LIN {X 106, Y 277, Z 59} c_vel
LIN {X 113, Y 269, Z 59} c_vel
LIN {X 118, Y 261, Z 59} c_vel
LIN {X 123, Y 253, Z 59} c_vel
LIN {X 127, Y 244, Z 59} c_vel
LIN {X 130, Y 235, Z 59} c_vel
LIN {X 131, Y 226, Z 59} c_vel
LIN {X 133, Y 217, Z 59} c_vel
LIN {X 133, Y 207, Z 59} c_vel
LIN {X 133, Y 197, Z 59} c_vel
LIN {X 131, Y 186, Z 59} c_vel
LIN {X 129, Y 173, Z 59} c_vel
LIN {X 126, Y 160, Z 59} c_vel
LIN {X 120, Y 138, Z 59} c_vel
LIN {X 115, Y 118, Z 59} c_vel
LIN {X 112, Y 106, Z 59} c_vel
LIN {X 111, Y 96, Z 59} c_vel
LIN {X 110, Y 88, Z 59} c_vel
LIN {X 110, Y 81, Z 59} c_vel
LIN {X 111, Y 74, Z 59} c_vel
LIN {X 113, Y 69, Z 59} c_vel
LIN {X 116, Y 63, Z 59} c_vel
LIN {X 119, Y 58, Z 59} c_vel
LIN {X 124, Y 53, Z 59} c_vel
LIN {X 130, Y 48, Z 59} c_vel
LIN {X 138, Y 43, Z 59} c_vel
LIN {X 111, Y 0, Z 59} c_vel
$OUT[4] = FALSE
WAIT SEC 10.0
LIN {X 111, Y 0, Z 60} c_vel
$OUT[4] = TRUE
LIN {X 111, Y 0, Z 60} c_vel
LIN {X 106, Y 3, Z 60} c_vel
LIN {X 97, Y 9, Z 60} c_vel
LIN {X 89, Y 16, Z 60} c_vel
LIN {X 83, Y 23, Z 60} c_vel
LIN {X 77, Y 31, Z 60} c_vel
LIN {X 71, Y 39, Z 60} c_vel
LIN {X 67, Y 47, Z 60} c_vel
LIN {X 64, Y 56, Z 60} c_vel
LIN {X 62, Y 64, Z 60} c_vel
LIN {X 60, Y 73, Z 60} c_vel
LIN {X 59, Y 82, Z 60} c_vel
LIN {X 59, Y 92, Z 60} c_vel
LIN {X 60, Y 103, Z 60} c_vel
LIN {X 62, Y 114, Z 60} c_vel
LIN {X 65, Y 127, Z 60} c_vel
LIN {X 69, Y 144, Z 60} c_vel
LIN {X 74, Y 163, Z 60} c_vel
LIN {X 79, Y 180, Z 60} c_vel
LIN {X 81, Y 191, Z 60} c_vel
LIN {X 82, Y 201, Z 60} c_vel
LIN {X 82, Y 209, Z 60} c_vel
LIN {X 82, Y 217, Z 60} c_vel
LIN {X 80, Y 223, Z 60} c_vel
LIN {X 78, Y 229, Z 60} c_vel
LIN {X 75, Y 234, Z 60} c_vel
LIN {X 71, Y 240, Z 60} c_vel
LIN {X 66, Y 245, Z 60} c_vel
LIN {X 60, Y 250, Z 60} c_vel
LIN {X 52, Y 256, Z 60} c_vel
LIN {X 42, Y 261, Z 60} c_vel
LIN {X 30, Y 267, Z 60} c_vel
LIN {X 16, Y 273, Z 60} c_vel
LIN {X 0, Y 278, Z 60} c_vel
LIN {X 14, Y 327, Z 60} c_vel
LIN {X 28, Y 322, Z 60} c_vel
LIN {X 43, Y 317, Z 60} c_vel
LIN {X 57, Y 311, Z 60} c_vel
LIN {X 70, Y 304, Z 60} c_vel
LIN {X 81, Y 298, Z 60} c_vel
LIN {X 90, Y 291, Z 60} c_vel
LIN {X 99, Y 284, Z 60} c_vel
LIN {X 106, Y 277, Z 60} c_vel
LIN {X 113, Y 269, Z 60} c_vel
LIN {X 118, Y 261, Z 60} c_vel
LIN {X 123, Y 253, Z 60} c_vel
LIN {X 127, Y 244, Z 60} c_vel
LIN {X 130, Y 235, Z 60} c_vel
LIN {X 131, Y 226, Z 60} c_vel
LIN {X 133, Y 217, Z 60} c_vel
LIN {X 133, Y 207, Z 60} c_vel
LIN {X 133, Y 197, Z 60} c_vel
LIN {X 131, Y 186, Z 60} c_vel
LIN {X 129, Y 173, Z 60} c_vel
LIN {X 126, Y 160, Z 60} c_vel
LIN {X 120, Y 138, Z 60} c_vel
LIN {X 115, Y 118, Z 60} c_vel
LIN {X 112, Y 106, Z 60} c_vel
LIN {X 111, Y 96, Z 60} c_vel
LIN {X 110, Y 88, Z 60} c_vel
LIN {X 110, Y 81, Z 60} c_vel
LIN {X 111, Y 74, Z 60} c_vel
LIN {X 113, Y 69, Z 60} c_vel
LIN {X 116, Y 63, Z 60} c_vel
LIN {X 119, Y 58, Z 60} c_vel
LIN {X 124, Y 53, Z 60} c_vel
LIN {X 130, Y 48, Z 60} c_vel
LIN {X 138, Y 43, Z 60} c_vel
LIN {X 111, Y 0, Z 60} c_vel
$OUT[4] = FALSE
WAIT SEC 10.0
LIN {X 111, Y 0, Z 61} c_vel
$OUT[4] = TRUE
LIN {X 111, Y 0, Z 61} c_vel
LIN {X 106, Y 3, Z 61} c_vel
LIN {X 97, Y 9, Z 61} c_vel
LIN {X 89, Y 16, Z 61} c_vel
LIN {X 83, Y 23, Z 61} c_vel
LIN {X 77, Y 31, Z 61} c_vel
LIN {X 71, Y 39, Z 61} c_vel
LIN {X 67, Y 47, Z 61} c_vel
LIN {X 64, Y 56, Z 61} c_vel
LIN {X 62, Y 64, Z 61} c_vel
LIN {X 60, Y 73, Z 61} c_vel
LIN {X 59, Y 82, Z 61} c_vel
LIN {X 59, Y 92, Z 61} c_vel
LIN {X 60, Y 103, Z 61} c_vel
LIN {X 62, Y 114, Z 61} c_vel
LIN {X 65, Y 127, Z 61} c_vel
LIN {X 69, Y 144, Z 61} c_vel
LIN {X 74, Y 163, Z 61} c_vel
LIN {X 79, Y 180, Z 61} c_vel
LIN {X 81, Y 191, Z 61} c_vel
LIN {X 82, Y 201, Z 61} c_vel
LIN {X 82, Y 209, Z 61} c_vel
LIN {X 82, Y 217, Z 61} c_vel
LIN {X 80, Y 223, Z 61} c_vel
LIN {X 78, Y 229, Z 61} c_vel
LIN {X 75, Y 234, Z 61} c_vel
LIN {X 71, Y 240, Z 61} c_vel
LIN {X 66, Y 245, Z 61} c_vel
LIN {X 60, Y 250, Z 61} c_vel
LIN {X 52, Y 256, Z 61} c_vel
LIN {X 42, Y 261, Z 61} c_vel
LIN {X 30, Y 267, Z 61} c_vel
LIN {X 16, Y 273, Z 61} c_vel
LIN {X 0, Y 278, Z 61} c_vel
LIN {X 14, Y 327, Z 61} c_vel
LIN {X 28, Y 322, Z 61} c_vel
LIN {X 43, Y 317, Z 61} c_vel
LIN {X 57, Y 311, Z 61} c_vel
LIN {X 70, Y 304, Z 61} c_vel
LIN {X 81, Y 298, Z 61} c_vel
LIN {X 90, Y 291, Z 61} c_vel
LIN {X 99, Y 284, Z 61} c_vel
LIN {X 106, Y 277, Z 61} c_vel
LIN {X 113, Y 269, Z 61} c_vel
LIN {X 118, Y 261, Z 61} c_vel
LIN {X 123, Y 253, Z 61} c_vel
LIN {X 127, Y 244, Z 61} c_vel
LIN {X 130, Y 235, Z 61} c_vel
LIN {X 131, Y 226, Z 61} c_vel
LIN {X 133, Y 217, Z 61} c_vel
LIN {X 133, Y 207, Z 61} c_vel
LIN {X 133, Y 197, Z 61} c_vel
LIN {X 131, Y 186, Z 61} c_vel
LIN {X 129, Y 173, Z 61} c_vel
LIN {X 126, Y 160, Z 61} c_vel
LIN {X 120, Y 138, Z 61} c_vel
LIN {X 115, Y 118, Z 61} c_vel
LIN {X 112, Y 106, Z 61} c_vel
LIN {X 111, Y 96, Z 61} c_vel
LIN {X 110, Y 88, Z 61} c_vel
LIN {X 110, Y 81, Z 61} c_vel
LIN {X 111, Y 74, Z 61} c_vel
LIN {X 113, Y 69, Z 61} c_vel
LIN {X 116, Y 63, Z 61} c_vel
LIN {X 119, Y 58, Z 61} c_vel
LIN {X 124, Y 53, Z 61} c_vel
LIN {X 130, Y 48, Z 61} c_vel
LIN {X 138, Y 43, Z 61} c_vel
LIN {X 111, Y 0, Z 61} c_vel
$OUT[4] = FALSE
WAIT SEC 10.0
LIN {X 111, Y 0, Z 62} c_vel
$OUT[4] = TRUE
LIN {X 111, Y 0, Z 62} c_vel
LIN {X 106, Y 3, Z 62} c_vel
LIN {X 97, Y 9, Z 62} c_vel
LIN {X 89, Y 16, Z 62} c_vel
LIN {X 83, Y 23, Z 62} c_vel
LIN {X 77, Y 31, Z 62} c_vel
LIN {X 71, Y 39, Z 62} c_vel
LIN {X 67, Y 47, Z 62} c_vel
LIN {X 64, Y 56, Z 62} c_vel
LIN {X 62, Y 64, Z 62} c_vel
LIN {X 60, Y 73, Z 62} c_vel
LIN {X 59, Y 82, Z 62} c_vel
LIN {X 59, Y 92, Z 62} c_vel
LIN {X 60, Y 103, Z 62} c_vel
LIN {X 62, Y 114, Z 62} c_vel
LIN {X 65, Y 127, Z 62} c_vel
LIN {X 69, Y 144, Z 62} c_vel
LIN {X 74, Y 163, Z 62} c_vel
LIN {X 79, Y 180, Z 62} c_vel
LIN {X 81, Y 191, Z 62} c_vel
LIN {X 82, Y 201, Z 62} c_vel
LIN {X 82, Y 209, Z 62} c_vel
LIN {X 82, Y 217, Z 62} c_vel
LIN {X 80, Y 223, Z 62} c_vel
LIN {X 78, Y 229, Z 62} c_vel
LIN {X 75, Y 234, Z 62} c_vel
LIN {X 71, Y 240, Z 62} c_vel
LIN {X 66, Y 245, Z 62} c_vel
LIN {X 60, Y 250, Z 62} c_vel
LIN {X 52, Y 256, Z 62} c_vel
LIN {X 42, Y 261, Z 62} c_vel
LIN {X 30, Y 267, Z 62} c_vel
LIN {X 16, Y 273, Z 62} c_vel
LIN {X 0, Y 278, Z 62} c_vel
LIN {X 14, Y 327, Z 62} c_vel
LIN {X 28, Y 322, Z 62} c_vel
LIN {X 43, Y 317, Z 62} c_vel
LIN {X 57, Y 311, Z 62} c_vel
LIN {X 70, Y 304, Z 62} c_vel
LIN {X 81, Y 298, Z 62} c_vel
LIN {X 90, Y 291, Z 62} c_vel
LIN {X 99, Y 284, Z 62} c_vel
LIN {X 106, Y 277, Z 62} c_vel
LIN {X 113, Y 269, Z 62} c_vel
LIN {X 118, Y 261, Z 62} c_vel
LIN {X 123, Y 253, Z 62} c_vel
LIN {X 127, Y 244, Z 62} c_vel
LIN {X 130, Y 235, Z 62} c_vel
LIN {X 131, Y 226, Z 62} c_vel
LIN {X 133, Y 217, Z 62} c_vel
LIN {X 133, Y 207, Z 62} c_vel
LIN {X 133, Y 197, Z 62} c_vel
LIN {X 131, Y 186, Z 62} c_vel
LIN {X 129, Y 173, Z 62} c_vel
LIN {X 126, Y 160, Z 62} c_vel
LIN {X 120, Y 138, Z 62} c_vel
LIN {X 115, Y 118, Z 62} c_vel
LIN {X 112, Y 106, Z 62} c_vel
LIN {X 111, Y 96, Z 62} c_vel
LIN {X 110, Y 88, Z 62} c_vel
LIN {X 110, Y 81, Z 62} c_vel
LIN {X 111, Y 74, Z 62} c_vel
LIN {X 113, Y 69, Z 62} c_vel
LIN {X 116, Y 63, Z 62} c_vel
LIN {X 119, Y 58, Z 62} c_vel
LIN {X 124, Y 53, Z 62} c_vel
LIN {X 130, Y 48, Z 62} c_vel
LIN {X 138, Y 43, Z 62} c_vel
LIN {X 111, Y 0, Z 62} c_vel
$OUT[4] = FALSE
WAIT SEC 10.0
LIN {X 111, Y 0, Z 63} c_vel
$OUT[4] = TRUE
LIN {X 111, Y 0, Z 63} c_vel
LIN {X 106, Y 3, Z 63} c_vel
LIN {X 97, Y 9, Z 63} c_vel
LIN {X 89, Y 16, Z 63} c_vel
LIN {X 83, Y 23, Z 63} c_vel
LIN {X 77, Y 31, Z 63} c_vel
LIN {X 71, Y 39, Z 63} c_vel
LIN {X 67, Y 47, Z 63} c_vel
LIN {X 64, Y 56, Z 63} c_vel
LIN {X 62, Y 64, Z 63} c_vel
LIN {X 60, Y 73, Z 63} c_vel
LIN {X 59, Y 82, Z 63} c_vel
LIN {X 59, Y 92, Z 63} c_vel
LIN {X 60, Y 103, Z 63} c_vel
LIN {X 62, Y 114, Z 63} c_vel
LIN {X 65, Y 127, Z 63} c_vel
LIN {X 69, Y 144, Z 63} c_vel
LIN {X 74, Y 163, Z 63} c_vel
LIN {X 79, Y 180, Z 63} c_vel
LIN {X 81, Y 191, Z 63} c_vel
LIN {X 82, Y 201, Z 63} c_vel
LIN {X 82, Y 209, Z 63} c_vel
LIN {X 82, Y 217, Z 63} c_vel
LIN {X 80, Y 223, Z 63} c_vel
LIN {X 78, Y 229, Z 63} c_vel
LIN {X 75, Y 234, Z 63} c_vel
LIN {X 71, Y 240, Z 63} c_vel
LIN {X 66, Y 245, Z 63} c_vel
LIN {X 60, Y 250, Z 63} c_vel
LIN {X 52, Y 256, Z 63} c_vel
LIN {X 42, Y 261, Z 63} c_vel
LIN {X 30, Y 267, Z 63} c_vel
LIN {X 16, Y 273, Z 63} c_vel
LIN {X 0, Y 278, Z 63} c_vel
LIN {X 14, Y 327, Z 63} c_vel
LIN {X 28, Y 322, Z 63} c_vel
LIN {X 43, Y 317, Z 63} c_vel
LIN {X 57, Y 311, Z 63} c_vel
LIN {X 70, Y 304, Z 63} c_vel
LIN {X 81, Y 298, Z 63} c_vel
LIN {X 90, Y 291, Z 63} c_vel
LIN {X 99, Y 284, Z 63} c_vel
LIN {X 106, Y 277, Z 63} c_vel
LIN {X 113, Y 269, Z 63} c_vel
LIN {X 118, Y 261, Z 63} c_vel
LIN {X 123, Y 253, Z 63} c_vel
LIN {X 127, Y 244, Z 63} c_vel
LIN {X 130, Y 235, Z 63} c_vel
LIN {X 131, Y 226, Z 63} c_vel
LIN {X 133, Y 217, Z 63} c_vel
LIN {X 133, Y 207, Z 63} c_vel
LIN {X 133, Y 197, Z 63} c_vel
LIN {X 131, Y 186, Z 63} c_vel
LIN {X 129, Y 173, Z 63} c_vel
LIN {X 126, Y 160, Z 63} c_vel
LIN {X 120, Y 138, Z 63} c_vel
LIN {X 115, Y 118, Z 63} c_vel
LIN {X 112, Y 106, Z 63} c_vel
LIN {X 111, Y 96, Z 63} c_vel
LIN {X 110, Y 88, Z 63} c_vel
LIN {X 110, Y 81, Z 63} c_vel
LIN {X 111, Y 74, Z 63} c_vel
LIN {X 113, Y 69, Z 63} c_vel
LIN {X 116, Y 63, Z 63} c_vel
LIN {X 119, Y 58, Z 63} c_vel
LIN {X 124, Y 53, Z 63} c_vel
LIN {X 130, Y 48, Z 63} c_vel
LIN {X 138, Y 43, Z 63} c_vel
LIN {X 111, Y 0, Z 63} c_vel
$OUT[4] = FALSE
WAIT SEC 10.0
LIN {X 111, Y 0, Z 64} c_vel
$OUT[4] = TRUE
LIN {X 111, Y 0, Z 64} c_vel
LIN {X 106, Y 3, Z 64} c_vel
LIN {X 97, Y 9, Z 64} c_vel
LIN {X 89, Y 16, Z 64} c_vel
LIN {X 83, Y 23, Z 64} c_vel
LIN {X 77, Y 31, Z 64} c_vel
LIN {X 71, Y 39, Z 64} c_vel
LIN {X 67, Y 47, Z 64} c_vel
LIN {X 64, Y 56, Z 64} c_vel
LIN {X 62, Y 64, Z 64} c_vel
LIN {X 60, Y 73, Z 64} c_vel
LIN {X 59, Y 82, Z 64} c_vel
LIN {X 59, Y 92, Z 64} c_vel
LIN {X 60, Y 103, Z 64} c_vel
LIN {X 62, Y 114, Z 64} c_vel
LIN {X 65, Y 127, Z 64} c_vel
LIN {X 69, Y 144, Z 64} c_vel
LIN {X 74, Y 163, Z 64} c_vel
LIN {X 79, Y 180, Z 64} c_vel
LIN {X 81, Y 191, Z 64} c_vel
LIN {X 82, Y 201, Z 64} c_vel
LIN {X 82, Y 209, Z 64} c_vel
LIN {X 82, Y 217, Z 64} c_vel
LIN {X 80, Y 223, Z 64} c_vel
LIN {X 78, Y 229, Z 64} c_vel
LIN {X 75, Y 234, Z 64} c_vel
LIN {X 71, Y 240, Z 64} c_vel
LIN {X 66, Y 245, Z 64} c_vel
LIN {X 60, Y 250, Z 64} c_vel
LIN {X 52, Y 256, Z 64} c_vel
LIN {X 42, Y 261, Z 64} c_vel
LIN {X 30, Y 267, Z 64} c_vel
LIN {X 16, Y 273, Z 64} c_vel
LIN {X 0, Y 278, Z 64} c_vel
LIN {X 14, Y 327, Z 64} c_vel
LIN {X 28, Y 322, Z 64} c_vel
LIN {X 43, Y 317, Z 64} c_vel
LIN {X 57, Y 311, Z 64} c_vel
LIN {X 70, Y 304, Z 64} c_vel
LIN {X 81, Y 298, Z 64} c_vel
LIN {X 90, Y 291, Z 64} c_vel
LIN {X 99, Y 284, Z 64} c_vel
LIN {X 106, Y 277, Z 64} c_vel
LIN {X 113, Y 269, Z 64} c_vel
LIN {X 118, Y 261, Z 64} c_vel
LIN {X 123, Y 253, Z 64} c_vel
LIN {X 127, Y 244, Z 64} c_vel
LIN {X 130, Y 235, Z 64} c_vel
LIN {X 131, Y 226, Z 64} c_vel
LIN {X 133, Y 217, Z 64} c_vel
LIN {X 133, Y 207, Z 64} c_vel
LIN {X 133, Y 197, Z 64} c_vel
LIN {X 131, Y 186, Z 64} c_vel
LIN {X 129, Y 173, Z 64} c_vel
LIN {X 126, Y 160, Z 64} c_vel
LIN {X 120, Y 138, Z 64} c_vel
LIN {X 115, Y 118, Z 64} c_vel
LIN {X 112, Y 106, Z 64} c_vel
LIN {X 111, Y 96, Z 64} c_vel
LIN {X 110, Y 88, Z 64} c_vel
LIN {X 110, Y 81, Z 64} c_vel
LIN {X 111, Y 74, Z 64} c_vel
LIN {X 113, Y 69, Z 64} c_vel
LIN {X 116, Y 63, Z 64} c_vel
LIN {X 119, Y 58, Z 64} c_vel
LIN {X 124, Y 53, Z 64} c_vel
LIN {X 130, Y 48, Z 64} c_vel
LIN {X 138, Y 43, Z 64} c_vel
LIN {X 111, Y 0, Z 64} c_vel
$OUT[4] = FALSE
WAIT SEC 10.0
LIN {X 111, Y 0, Z 65} c_vel
$OUT[4] = TRUE
LIN {X 111, Y 0, Z 65} c_vel
LIN {X 106, Y 3, Z 65} c_vel
LIN {X 97, Y 9, Z 65} c_vel
LIN {X 89, Y 16, Z 65} c_vel
LIN {X 83, Y 23, Z 65} c_vel
LIN {X 77, Y 31, Z 65} c_vel
LIN {X 71, Y 39, Z 65} c_vel
LIN {X 67, Y 47, Z 65} c_vel
LIN {X 64, Y 56, Z 65} c_vel
LIN {X 62, Y 64, Z 65} c_vel
LIN {X 60, Y 73, Z 65} c_vel
LIN {X 59, Y 82, Z 65} c_vel
LIN {X 59, Y 92, Z 65} c_vel
LIN {X 60, Y 103, Z 65} c_vel
LIN {X 62, Y 114, Z 65} c_vel
LIN {X 65, Y 127, Z 65} c_vel
LIN {X 69, Y 144, Z 65} c_vel
LIN {X 74, Y 163, Z 65} c_vel
LIN {X 79, Y 180, Z 65} c_vel
LIN {X 81, Y 191, Z 65} c_vel
LIN {X 82, Y 201, Z 65} c_vel
LIN {X 82, Y 209, Z 65} c_vel
LIN {X 82, Y 217, Z 65} c_vel
LIN {X 80, Y 223, Z 65} c_vel
LIN {X 78, Y 229, Z 65} c_vel
LIN {X 75, Y 234, Z 65} c_vel
LIN {X 71, Y 240, Z 65} c_vel
LIN {X 66, Y 245, Z 65} c_vel
LIN {X 60, Y 250, Z 65} c_vel
LIN {X 52, Y 256, Z 65} c_vel
LIN {X 42, Y 261, Z 65} c_vel
LIN {X 30, Y 267, Z 65} c_vel
LIN {X 16, Y 273, Z 65} c_vel
LIN {X 0, Y 278, Z 65} c_vel
LIN {X 14, Y 327, Z 65} c_vel
LIN {X 28, Y 322, Z 65} c_vel
LIN {X 43, Y 317, Z 65} c_vel
LIN {X 57, Y 311, Z 65} c_vel
LIN {X 70, Y 304, Z 65} c_vel
LIN {X 81, Y 298, Z 65} c_vel
LIN {X 90, Y 291, Z 65} c_vel
LIN {X 99, Y 284, Z 65} c_vel
LIN {X 106, Y 277, Z 65} c_vel
LIN {X 113, Y 269, Z 65} c_vel
LIN {X 118, Y 261, Z 65} c_vel
LIN {X 123, Y 253, Z 65} c_vel
LIN {X 127, Y 244, Z 65} c_vel
LIN {X 130, Y 235, Z 65} c_vel
LIN {X 131, Y 226, Z 65} c_vel
LIN {X 133, Y 217, Z 65} c_vel
LIN {X 133, Y 207, Z 65} c_vel
LIN {X 133, Y 197, Z 65} c_vel
LIN {X 131, Y 186, Z 65} c_vel
LIN {X 129, Y 173, Z 65} c_vel
LIN {X 126, Y 160, Z 65} c_vel
LIN {X 120, Y 138, Z 65} c_vel
LIN {X 115, Y 118, Z 65} c_vel
LIN {X 112, Y 106, Z 65} c_vel
LIN {X 111, Y 96, Z 65} c_vel
LIN {X 110, Y 88, Z 65} c_vel
LIN {X 110, Y 81, Z 65} c_vel
LIN {X 111, Y 74, Z 65} c_vel
LIN {X 113, Y 69, Z 65} c_vel
LIN {X 116, Y 63, Z 65} c_vel
LIN {X 119, Y 58, Z 65} c_vel
LIN {X 124, Y 53, Z 65} c_vel
LIN {X 130, Y 48, Z 65} c_vel
LIN {X 138, Y 43, Z 65} c_vel
LIN {X 111, Y 0, Z 65} c_vel
$OUT[4] = FALSE
WAIT SEC 10.0
LIN {X 111, Y 0, Z 66} c_vel
$OUT[4] = TRUE
LIN {X 111, Y 0, Z 66} c_vel
LIN {X 106, Y 3, Z 66} c_vel
LIN {X 97, Y 9, Z 66} c_vel
LIN {X 89, Y 16, Z 66} c_vel
LIN {X 83, Y 23, Z 66} c_vel
LIN {X 77, Y 31, Z 66} c_vel
LIN {X 71, Y 39, Z 66} c_vel
LIN {X 67, Y 47, Z 66} c_vel
LIN {X 64, Y 56, Z 66} c_vel
LIN {X 62, Y 64, Z 66} c_vel
LIN {X 60, Y 73, Z 66} c_vel
LIN {X 59, Y 82, Z 66} c_vel
LIN {X 59, Y 92, Z 66} c_vel
LIN {X 60, Y 103, Z 66} c_vel
LIN {X 62, Y 114, Z 66} c_vel
LIN {X 65, Y 127, Z 66} c_vel
LIN {X 69, Y 144, Z 66} c_vel
LIN {X 74, Y 163, Z 66} c_vel
LIN {X 79, Y 180, Z 66} c_vel
LIN {X 81, Y 191, Z 66} c_vel
LIN {X 82, Y 201, Z 66} c_vel
LIN {X 82, Y 209, Z 66} c_vel
LIN {X 82, Y 217, Z 66} c_vel
LIN {X 80, Y 223, Z 66} c_vel
LIN {X 78, Y 229, Z 66} c_vel
LIN {X 75, Y 234, Z 66} c_vel
LIN {X 71, Y 240, Z 66} c_vel
LIN {X 66, Y 245, Z 66} c_vel
LIN {X 60, Y 250, Z 66} c_vel
LIN {X 52, Y 256, Z 66} c_vel
LIN {X 42, Y 261, Z 66} c_vel
LIN {X 30, Y 267, Z 66} c_vel
LIN {X 16, Y 273, Z 66} c_vel
LIN {X 0, Y 278, Z 66} c_vel
LIN {X 14, Y 327, Z 66} c_vel
LIN {X 28, Y 322, Z 66} c_vel
LIN {X 43, Y 317, Z 66} c_vel
LIN {X 57, Y 311, Z 66} c_vel
LIN {X 70, Y 304, Z 66} c_vel
LIN {X 81, Y 298, Z 66} c_vel
LIN {X 90, Y 291, Z 66} c_vel
LIN {X 99, Y 284, Z 66} c_vel
LIN {X 106, Y 277, Z 66} c_vel
LIN {X 113, Y 269, Z 66} c_vel
LIN {X 118, Y 261, Z 66} c_vel
LIN {X 123, Y 253, Z 66} c_vel
LIN {X 127, Y 244, Z 66} c_vel
LIN {X 130, Y 235, Z 66} c_vel
LIN {X 131, Y 226, Z 66} c_vel
LIN {X 133, Y 217, Z 66} c_vel
LIN {X 133, Y 207, Z 66} c_vel
LIN {X 133, Y 197, Z 66} c_vel
LIN {X 131, Y 186, Z 66} c_vel
LIN {X 129, Y 173, Z 66} c_vel
LIN {X 126, Y 160, Z 66} c_vel
LIN {X 120, Y 138, Z 66} c_vel
LIN {X 115, Y 118, Z 66} c_vel
LIN {X 112, Y 106, Z 66} c_vel
LIN {X 111, Y 96, Z 66} c_vel
LIN {X 110, Y 88, Z 66} c_vel
LIN {X 110, Y 81, Z 66} c_vel
LIN {X 111, Y 74, Z 66} c_vel
LIN {X 113, Y 69, Z 66} c_vel
LIN {X 116, Y 63, Z 66} c_vel
LIN {X 119, Y 58, Z 66} c_vel
LIN {X 124, Y 53, Z 66} c_vel
LIN {X 130, Y 48, Z 66} c_vel
LIN {X 138, Y 43, Z 66} c_vel
LIN {X 111, Y 0, Z 66} c_vel
$OUT[4] = FALSE
WAIT SEC 10.0
LIN {X 111, Y 0, Z 67} c_vel
$OUT[4] = TRUE
LIN {X 111, Y 0, Z 67} c_vel
LIN {X 106, Y 3, Z 67} c_vel
LIN {X 97, Y 9, Z 67} c_vel
LIN {X 89, Y 16, Z 67} c_vel
LIN {X 83, Y 23, Z 67} c_vel
LIN {X 77, Y 31, Z 67} c_vel
LIN {X 71, Y 39, Z 67} c_vel
LIN {X 67, Y 47, Z 67} c_vel
LIN {X 64, Y 56, Z 67} c_vel
LIN {X 62, Y 64, Z 67} c_vel
LIN {X 60, Y 73, Z 67} c_vel
LIN {X 59, Y 82, Z 67} c_vel
LIN {X 59, Y 91, Z 67} c_vel
LIN {X 59, Y 92, Z 67} c_vel
LIN {X 60, Y 103, Z 67} c_vel
LIN {X 62, Y 114, Z 67} c_vel
LIN {X 65, Y 127, Z 67} c_vel
LIN {X 69, Y 144, Z 67} c_vel
LIN {X 74, Y 163, Z 67} c_vel
LIN {X 79, Y 180, Z 67} c_vel
LIN {X 81, Y 191, Z 67} c_vel
LIN {X 82, Y 201, Z 67} c_vel
LIN {X 82, Y 209, Z 67} c_vel
LIN {X 82, Y 217, Z 67} c_vel
LIN {X 80, Y 223, Z 67} c_vel
LIN {X 78, Y 229, Z 67} c_vel
LIN {X 75, Y 234, Z 67} c_vel
LIN {X 71, Y 240, Z 67} c_vel
LIN {X 66, Y 245, Z 67} c_vel
LIN {X 60, Y 250, Z 67} c_vel
LIN {X 52, Y 256, Z 67} c_vel
LIN {X 42, Y 261, Z 67} c_vel
LIN {X 30, Y 267, Z 67} c_vel
LIN {X 16, Y 273, Z 67} c_vel
LIN {X 0, Y 278, Z 67} c_vel
LIN {X 14, Y 327, Z 67} c_vel
LIN {X 28, Y 322, Z 67} c_vel
LIN {X 43, Y 317, Z 67} c_vel
LIN {X 57, Y 311, Z 67} c_vel
LIN {X 70, Y 304, Z 67} c_vel
LIN {X 81, Y 298, Z 67} c_vel
LIN {X 90, Y 291, Z 67} c_vel
LIN {X 99, Y 284, Z 67} c_vel
LIN {X 106, Y 277, Z 67} c_vel
LIN {X 113, Y 269, Z 67} c_vel
LIN {X 118, Y 261, Z 67} c_vel
LIN {X 123, Y 253, Z 67} c_vel
LIN {X 127, Y 244, Z 67} c_vel
LIN {X 130, Y 235, Z 67} c_vel
LIN {X 131, Y 226, Z 67} c_vel
LIN {X 133, Y 217, Z 67} c_vel
LIN {X 133, Y 207, Z 67} c_vel
LIN {X 133, Y 197, Z 67} c_vel
LIN {X 131, Y 186, Z 67} c_vel
LIN {X 129, Y 173, Z 67} c_vel
LIN {X 126, Y 160, Z 67} c_vel
LIN {X 120, Y 138, Z 67} c_vel
LIN {X 115, Y 118, Z 67} c_vel
LIN {X 112, Y 106, Z 67} c_vel
LIN {X 111, Y 96, Z 67} c_vel
LIN {X 110, Y 88, Z 67} c_vel
LIN {X 110, Y 81, Z 67} c_vel
LIN {X 111, Y 74, Z 67} c_vel
LIN {X 113, Y 69, Z 67} c_vel
LIN {X 116, Y 63, Z 67} c_vel
LIN {X 119, Y 58, Z 67} c_vel
LIN {X 124, Y 53, Z 67} c_vel
LIN {X 130, Y 48, Z 67} c_vel
LIN {X 138, Y 43, Z 67} c_vel
LIN {X 111, Y 0, Z 67} c_vel
$OUT[4] = FALSE
WAIT SEC 10.0
LIN {X 111, Y 0, Z 68} c_vel
$OUT[4] = TRUE
LIN {X 111, Y 0, Z 68} c_vel
LIN {X 106, Y 3, Z 68} c_vel
LIN {X 97, Y 9, Z 68} c_vel
LIN {X 89, Y 16, Z 68} c_vel
LIN {X 83, Y 23, Z 68} c_vel
LIN {X 77, Y 31, Z 68} c_vel
LIN {X 71, Y 39, Z 68} c_vel
LIN {X 67, Y 47, Z 68} c_vel
LIN {X 64, Y 56, Z 68} c_vel
LIN {X 62, Y 64, Z 68} c_vel
LIN {X 60, Y 73, Z 68} c_vel
LIN {X 59, Y 82, Z 68} c_vel
LIN {X 59, Y 91, Z 68} c_vel
LIN {X 59, Y 92, Z 68} c_vel
LIN {X 60, Y 103, Z 68} c_vel
LIN {X 62, Y 114, Z 68} c_vel
LIN {X 65, Y 127, Z 68} c_vel
LIN {X 69, Y 144, Z 68} c_vel
LIN {X 74, Y 163, Z 68} c_vel
LIN {X 79, Y 180, Z 68} c_vel
LIN {X 81, Y 191, Z 68} c_vel
LIN {X 82, Y 201, Z 68} c_vel
LIN {X 82, Y 209, Z 68} c_vel
LIN {X 82, Y 217, Z 68} c_vel
LIN {X 80, Y 223, Z 68} c_vel
LIN {X 78, Y 229, Z 68} c_vel
LIN {X 75, Y 234, Z 68} c_vel
LIN {X 71, Y 240, Z 68} c_vel
LIN {X 66, Y 245, Z 68} c_vel
LIN {X 60, Y 250, Z 68} c_vel
LIN {X 52, Y 256, Z 68} c_vel
LIN {X 42, Y 261, Z 68} c_vel
LIN {X 30, Y 267, Z 68} c_vel
LIN {X 16, Y 273, Z 68} c_vel
LIN {X 0, Y 278, Z 68} c_vel
LIN {X 14, Y 327, Z 68} c_vel
LIN {X 28, Y 322, Z 68} c_vel
LIN {X 43, Y 317, Z 68} c_vel
LIN {X 57, Y 311, Z 68} c_vel
LIN {X 70, Y 304, Z 68} c_vel
LIN {X 81, Y 298, Z 68} c_vel
LIN {X 90, Y 291, Z 68} c_vel
LIN {X 99, Y 284, Z 68} c_vel
LIN {X 106, Y 277, Z 68} c_vel
LIN {X 113, Y 269, Z 68} c_vel
LIN {X 118, Y 261, Z 68} c_vel
LIN {X 123, Y 253, Z 68} c_vel
LIN {X 127, Y 244, Z 68} c_vel
LIN {X 130, Y 235, Z 68} c_vel
LIN {X 131, Y 226, Z 68} c_vel
LIN {X 133, Y 217, Z 68} c_vel
LIN {X 133, Y 207, Z 68} c_vel
LIN {X 133, Y 197, Z 68} c_vel
LIN {X 131, Y 186, Z 68} c_vel
LIN {X 129, Y 173, Z 68} c_vel
LIN {X 126, Y 160, Z 68} c_vel
LIN {X 120, Y 138, Z 68} c_vel
LIN {X 115, Y 118, Z 68} c_vel
LIN {X 112, Y 106, Z 68} c_vel
LIN {X 111, Y 96, Z 68} c_vel
LIN {X 110, Y 88, Z 68} c_vel
LIN {X 110, Y 81, Z 68} c_vel
LIN {X 111, Y 74, Z 68} c_vel
LIN {X 113, Y 69, Z 68} c_vel
LIN {X 116, Y 63, Z 68} c_vel
LIN {X 119, Y 58, Z 68} c_vel
LIN {X 124, Y 53, Z 68} c_vel
LIN {X 130, Y 48, Z 68} c_vel
LIN {X 138, Y 43, Z 68} c_vel
LIN {X 111, Y 0, Z 68} c_vel
$OUT[4] = FALSE
WAIT SEC 10.0
LIN {X 111, Y 0, Z 69} c_vel
$OUT[4] = TRUE
LIN {X 111, Y 0, Z 69} c_vel
LIN {X 106, Y 3, Z 69} c_vel
LIN {X 97, Y 9, Z 69} c_vel
LIN {X 89, Y 16, Z 69} c_vel
LIN {X 83, Y 23, Z 69} c_vel
LIN {X 77, Y 31, Z 69} c_vel
LIN {X 71, Y 39, Z 69} c_vel
LIN {X 67, Y 47, Z 69} c_vel
LIN {X 64, Y 56, Z 69} c_vel
LIN {X 62, Y 64, Z 69} c_vel
LIN {X 60, Y 73, Z 69} c_vel
LIN {X 59, Y 82, Z 69} c_vel
LIN {X 59, Y 92, Z 69} c_vel
LIN {X 60, Y 103, Z 69} c_vel
LIN {X 62, Y 114, Z 69} c_vel
LIN {X 65, Y 127, Z 69} c_vel
LIN {X 69, Y 144, Z 69} c_vel
LIN {X 74, Y 163, Z 69} c_vel
LIN {X 79, Y 180, Z 69} c_vel
LIN {X 81, Y 191, Z 69} c_vel
LIN {X 82, Y 201, Z 69} c_vel
LIN {X 82, Y 209, Z 69} c_vel
LIN {X 82, Y 217, Z 69} c_vel
LIN {X 80, Y 223, Z 69} c_vel
LIN {X 78, Y 229, Z 69} c_vel
LIN {X 75, Y 234, Z 69} c_vel
LIN {X 71, Y 240, Z 69} c_vel
LIN {X 66, Y 245, Z 69} c_vel
LIN {X 60, Y 250, Z 69} c_vel
LIN {X 52, Y 256, Z 69} c_vel
LIN {X 42, Y 261, Z 69} c_vel
LIN {X 30, Y 267, Z 69} c_vel
LIN {X 16, Y 273, Z 69} c_vel
LIN {X 0, Y 278, Z 69} c_vel
LIN {X 14, Y 327, Z 69} c_vel
LIN {X 28, Y 322, Z 69} c_vel
LIN {X 43, Y 317, Z 69} c_vel
LIN {X 57, Y 311, Z 69} c_vel
LIN {X 70, Y 304, Z 69} c_vel
LIN {X 81, Y 298, Z 69} c_vel
LIN {X 90, Y 291, Z 69} c_vel
LIN {X 99, Y 284, Z 69} c_vel
LIN {X 106, Y 277, Z 69} c_vel
LIN {X 113, Y 269, Z 69} c_vel
LIN {X 118, Y 261, Z 69} c_vel
LIN {X 123, Y 253, Z 69} c_vel
LIN {X 127, Y 244, Z 69} c_vel
LIN {X 130, Y 235, Z 69} c_vel
LIN {X 131, Y 226, Z 69} c_vel
LIN {X 133, Y 217, Z 69} c_vel
LIN {X 133, Y 207, Z 69} c_vel
LIN {X 133, Y 197, Z 69} c_vel
LIN {X 131, Y 186, Z 69} c_vel
LIN {X 129, Y 173, Z 69} c_vel
LIN {X 126, Y 160, Z 69} c_vel
LIN {X 120, Y 138, Z 69} c_vel
LIN {X 115, Y 118, Z 69} c_vel
LIN {X 112, Y 106, Z 69} c_vel
LIN {X 111, Y 96, Z 69} c_vel
LIN {X 110, Y 88, Z 69} c_vel
LIN {X 110, Y 81, Z 69} c_vel
LIN {X 111, Y 74, Z 69} c_vel
LIN {X 113, Y 69, Z 69} c_vel
LIN {X 116, Y 63, Z 69} c_vel
LIN {X 119, Y 58, Z 69} c_vel
LIN {X 124, Y 53, Z 69} c_vel
LIN {X 130, Y 48, Z 69} c_vel
LIN {X 138, Y 43, Z 69} c_vel
LIN {X 111, Y 0, Z 69} c_vel
$OUT[4] = FALSE
WAIT SEC 10.0
LIN {X 111, Y 0, Z 70} c_vel
$OUT[4] = TRUE
LIN {X 111, Y 0, Z 70} c_vel
LIN {X 106, Y 3, Z 70} c_vel
LIN {X 97, Y 9, Z 70} c_vel
LIN {X 89, Y 16, Z 70} c_vel
LIN {X 83, Y 23, Z 70} c_vel
LIN {X 77, Y 31, Z 70} c_vel
LIN {X 71, Y 39, Z 70} c_vel
LIN {X 67, Y 47, Z 70} c_vel
LIN {X 64, Y 56, Z 70} c_vel
LIN {X 62, Y 64, Z 70} c_vel
LIN {X 60, Y 73, Z 70} c_vel
LIN {X 59, Y 82, Z 70} c_vel
LIN {X 59, Y 92, Z 70} c_vel
LIN {X 60, Y 103, Z 70} c_vel
LIN {X 62, Y 114, Z 70} c_vel
LIN {X 65, Y 127, Z 70} c_vel
LIN {X 69, Y 144, Z 70} c_vel
LIN {X 74, Y 163, Z 70} c_vel
LIN {X 79, Y 180, Z 70} c_vel
LIN {X 81, Y 191, Z 70} c_vel
LIN {X 82, Y 201, Z 70} c_vel
LIN {X 82, Y 209, Z 70} c_vel
LIN {X 82, Y 217, Z 70} c_vel
LIN {X 80, Y 223, Z 70} c_vel
LIN {X 78, Y 229, Z 70} c_vel
LIN {X 75, Y 234, Z 70} c_vel
LIN {X 71, Y 240, Z 70} c_vel
LIN {X 66, Y 245, Z 70} c_vel
LIN {X 60, Y 250, Z 70} c_vel
LIN {X 52, Y 256, Z 70} c_vel
LIN {X 42, Y 261, Z 70} c_vel
LIN {X 30, Y 267, Z 70} c_vel
LIN {X 16, Y 273, Z 70} c_vel
LIN {X 0, Y 278, Z 70} c_vel
LIN {X 14, Y 327, Z 70} c_vel
LIN {X 28, Y 322, Z 70} c_vel
LIN {X 43, Y 317, Z 70} c_vel
LIN {X 57, Y 311, Z 70} c_vel
LIN {X 70, Y 304, Z 70} c_vel
LIN {X 81, Y 298, Z 70} c_vel
LIN {X 90, Y 291, Z 70} c_vel
LIN {X 99, Y 284, Z 70} c_vel
LIN {X 106, Y 277, Z 70} c_vel
LIN {X 113, Y 269, Z 70} c_vel
LIN {X 118, Y 261, Z 70} c_vel
LIN {X 123, Y 253, Z 70} c_vel
LIN {X 127, Y 244, Z 70} c_vel
LIN {X 130, Y 235, Z 70} c_vel
LIN {X 131, Y 226, Z 70} c_vel
LIN {X 133, Y 217, Z 70} c_vel
LIN {X 133, Y 207, Z 70} c_vel
LIN {X 133, Y 197, Z 70} c_vel
LIN {X 131, Y 186, Z 70} c_vel
LIN {X 129, Y 173, Z 70} c_vel
LIN {X 126, Y 160, Z 70} c_vel
LIN {X 120, Y 138, Z 70} c_vel
LIN {X 115, Y 118, Z 70} c_vel
LIN {X 112, Y 106, Z 70} c_vel
LIN {X 111, Y 96, Z 70} c_vel
LIN {X 110, Y 88, Z 70} c_vel
LIN {X 110, Y 81, Z 70} c_vel
LIN {X 111, Y 74, Z 70} c_vel
LIN {X 113, Y 69, Z 70} c_vel
LIN {X 116, Y 63, Z 70} c_vel
LIN {X 119, Y 58, Z 70} c_vel
LIN {X 124, Y 53, Z 70} c_vel
LIN {X 130, Y 48, Z 70} c_vel
LIN {X 138, Y 43, Z 70} c_vel
LIN {X 111, Y 0, Z 70} c_vel
$OUT[4] = FALSE
WAIT SEC 10.0
LIN {X 111, Y 0, Z 71} c_vel
$OUT[4] = TRUE
LIN {X 111, Y 0, Z 71} c_vel
LIN {X 106, Y 3, Z 71} c_vel
LIN {X 97, Y 9, Z 71} c_vel
LIN {X 89, Y 16, Z 71} c_vel
LIN {X 83, Y 23, Z 71} c_vel
LIN {X 77, Y 31, Z 71} c_vel
LIN {X 71, Y 39, Z 71} c_vel
LIN {X 67, Y 47, Z 71} c_vel
LIN {X 64, Y 56, Z 71} c_vel
LIN {X 62, Y 64, Z 71} c_vel
LIN {X 60, Y 73, Z 71} c_vel
LIN {X 59, Y 82, Z 71} c_vel
LIN {X 59, Y 92, Z 71} c_vel
LIN {X 60, Y 103, Z 71} c_vel
LIN {X 62, Y 114, Z 71} c_vel
LIN {X 65, Y 127, Z 71} c_vel
LIN {X 69, Y 144, Z 71} c_vel
LIN {X 74, Y 163, Z 71} c_vel
LIN {X 79, Y 180, Z 71} c_vel
LIN {X 81, Y 191, Z 71} c_vel
LIN {X 82, Y 201, Z 71} c_vel
LIN {X 82, Y 209, Z 71} c_vel
LIN {X 82, Y 217, Z 71} c_vel
LIN {X 80, Y 223, Z 71} c_vel
LIN {X 78, Y 229, Z 71} c_vel
LIN {X 75, Y 234, Z 71} c_vel
LIN {X 71, Y 240, Z 71} c_vel
LIN {X 66, Y 245, Z 71} c_vel
LIN {X 60, Y 250, Z 71} c_vel
LIN {X 52, Y 256, Z 71} c_vel
LIN {X 42, Y 261, Z 71} c_vel
LIN {X 30, Y 267, Z 71} c_vel
LIN {X 16, Y 273, Z 71} c_vel
LIN {X 0, Y 278, Z 71} c_vel
LIN {X 14, Y 327, Z 71} c_vel
LIN {X 28, Y 322, Z 71} c_vel
LIN {X 43, Y 317, Z 71} c_vel
LIN {X 57, Y 311, Z 71} c_vel
LIN {X 70, Y 304, Z 71} c_vel
LIN {X 81, Y 298, Z 71} c_vel
LIN {X 90, Y 291, Z 71} c_vel
LIN {X 99, Y 284, Z 71} c_vel
LIN {X 106, Y 277, Z 71} c_vel
LIN {X 113, Y 269, Z 71} c_vel
LIN {X 118, Y 261, Z 71} c_vel
LIN {X 123, Y 253, Z 71} c_vel
LIN {X 127, Y 244, Z 71} c_vel
LIN {X 130, Y 235, Z 71} c_vel
LIN {X 131, Y 226, Z 71} c_vel
LIN {X 133, Y 217, Z 71} c_vel
LIN {X 133, Y 207, Z 71} c_vel
LIN {X 133, Y 197, Z 71} c_vel
LIN {X 131, Y 186, Z 71} c_vel
LIN {X 129, Y 173, Z 71} c_vel
LIN {X 126, Y 160, Z 71} c_vel
LIN {X 120, Y 138, Z 71} c_vel
LIN {X 115, Y 118, Z 71} c_vel
LIN {X 112, Y 106, Z 71} c_vel
LIN {X 111, Y 96, Z 71} c_vel
LIN {X 110, Y 88, Z 71} c_vel
LIN {X 110, Y 81, Z 71} c_vel
LIN {X 111, Y 74, Z 71} c_vel
LIN {X 113, Y 69, Z 71} c_vel
LIN {X 116, Y 63, Z 71} c_vel
LIN {X 119, Y 58, Z 71} c_vel
LIN {X 124, Y 53, Z 71} c_vel
LIN {X 130, Y 48, Z 71} c_vel
LIN {X 138, Y 43, Z 71} c_vel
LIN {X 111, Y 0, Z 71} c_vel
$OUT[4] = FALSE
WAIT SEC 10.0
LIN {X 111, Y 0, Z 72} c_vel
$OUT[4] = TRUE
LIN {X 111, Y 0, Z 72} c_vel
LIN {X 106, Y 3, Z 72} c_vel
LIN {X 97, Y 9, Z 72} c_vel
LIN {X 89, Y 16, Z 72} c_vel
LIN {X 83, Y 23, Z 72} c_vel
LIN {X 77, Y 31, Z 72} c_vel
LIN {X 71, Y 39, Z 72} c_vel
LIN {X 67, Y 47, Z 72} c_vel
LIN {X 64, Y 56, Z 72} c_vel
LIN {X 62, Y 64, Z 72} c_vel
LIN {X 60, Y 73, Z 72} c_vel
LIN {X 59, Y 82, Z 72} c_vel
LIN {X 59, Y 92, Z 72} c_vel
LIN {X 60, Y 103, Z 72} c_vel
LIN {X 62, Y 114, Z 72} c_vel
LIN {X 65, Y 127, Z 72} c_vel
LIN {X 69, Y 144, Z 72} c_vel
LIN {X 74, Y 163, Z 72} c_vel
LIN {X 79, Y 180, Z 72} c_vel
LIN {X 81, Y 191, Z 72} c_vel
LIN {X 82, Y 201, Z 72} c_vel
LIN {X 82, Y 209, Z 72} c_vel
LIN {X 82, Y 217, Z 72} c_vel
LIN {X 80, Y 223, Z 72} c_vel
LIN {X 78, Y 229, Z 72} c_vel
LIN {X 75, Y 234, Z 72} c_vel
LIN {X 71, Y 240, Z 72} c_vel
LIN {X 66, Y 245, Z 72} c_vel
LIN {X 60, Y 250, Z 72} c_vel
LIN {X 52, Y 256, Z 72} c_vel
LIN {X 42, Y 261, Z 72} c_vel
LIN {X 30, Y 267, Z 72} c_vel
LIN {X 16, Y 273, Z 72} c_vel
LIN {X 0, Y 278, Z 72} c_vel
LIN {X 14, Y 327, Z 72} c_vel
LIN {X 28, Y 322, Z 72} c_vel
LIN {X 43, Y 317, Z 72} c_vel
LIN {X 57, Y 311, Z 72} c_vel
LIN {X 70, Y 304, Z 72} c_vel
LIN {X 81, Y 298, Z 72} c_vel
LIN {X 90, Y 291, Z 72} c_vel
LIN {X 99, Y 284, Z 72} c_vel
LIN {X 106, Y 277, Z 72} c_vel
LIN {X 113, Y 269, Z 72} c_vel
LIN {X 118, Y 261, Z 72} c_vel
LIN {X 123, Y 253, Z 72} c_vel
LIN {X 127, Y 244, Z 72} c_vel
LIN {X 130, Y 235, Z 72} c_vel
LIN {X 131, Y 226, Z 72} c_vel
LIN {X 133, Y 217, Z 72} c_vel
LIN {X 133, Y 207, Z 72} c_vel
LIN {X 133, Y 197, Z 72} c_vel
LIN {X 131, Y 186, Z 72} c_vel
LIN {X 129, Y 173, Z 72} c_vel
LIN {X 126, Y 160, Z 72} c_vel
LIN {X 120, Y 138, Z 72} c_vel
LIN {X 115, Y 118, Z 72} c_vel
LIN {X 112, Y 106, Z 72} c_vel
LIN {X 111, Y 96, Z 72} c_vel
LIN {X 110, Y 88, Z 72} c_vel
LIN {X 110, Y 81, Z 72} c_vel
LIN {X 111, Y 74, Z 72} c_vel
LIN {X 113, Y 69, Z 72} c_vel
LIN {X 116, Y 63, Z 72} c_vel
LIN {X 119, Y 58, Z 72} c_vel
LIN {X 124, Y 53, Z 72} c_vel
LIN {X 130, Y 48, Z 72} c_vel
LIN {X 138, Y 43, Z 72} c_vel
LIN {X 111, Y 0, Z 72} c_vel
$OUT[4] = FALSE
WAIT SEC 10.0
LIN {X 111, Y 0, Z 73} c_vel
$OUT[4] = TRUE
LIN {X 111, Y 0, Z 73} c_vel
LIN {X 106, Y 3, Z 73} c_vel
LIN {X 97, Y 9, Z 73} c_vel
LIN {X 89, Y 16, Z 73} c_vel
LIN {X 83, Y 23, Z 73} c_vel
LIN {X 77, Y 31, Z 73} c_vel
LIN {X 71, Y 39, Z 73} c_vel
LIN {X 67, Y 47, Z 73} c_vel
LIN {X 64, Y 56, Z 73} c_vel
LIN {X 62, Y 64, Z 73} c_vel
LIN {X 60, Y 73, Z 73} c_vel
LIN {X 59, Y 82, Z 73} c_vel
LIN {X 59, Y 92, Z 73} c_vel
LIN {X 60, Y 103, Z 73} c_vel
LIN {X 62, Y 114, Z 73} c_vel
LIN {X 65, Y 127, Z 73} c_vel
LIN {X 69, Y 144, Z 73} c_vel
LIN {X 74, Y 163, Z 73} c_vel
LIN {X 79, Y 180, Z 73} c_vel
LIN {X 81, Y 191, Z 73} c_vel
LIN {X 82, Y 201, Z 73} c_vel
LIN {X 82, Y 209, Z 73} c_vel
LIN {X 82, Y 217, Z 73} c_vel
LIN {X 80, Y 223, Z 73} c_vel
LIN {X 78, Y 229, Z 73} c_vel
LIN {X 75, Y 234, Z 73} c_vel
LIN {X 71, Y 240, Z 73} c_vel
LIN {X 66, Y 245, Z 73} c_vel
LIN {X 60, Y 250, Z 73} c_vel
LIN {X 52, Y 256, Z 73} c_vel
LIN {X 42, Y 261, Z 73} c_vel
LIN {X 30, Y 267, Z 73} c_vel
LIN {X 16, Y 273, Z 73} c_vel
LIN {X 0, Y 278, Z 73} c_vel
LIN {X 14, Y 327, Z 73} c_vel
LIN {X 28, Y 322, Z 73} c_vel
LIN {X 43, Y 317, Z 73} c_vel
LIN {X 57, Y 311, Z 73} c_vel
LIN {X 70, Y 304, Z 73} c_vel
LIN {X 81, Y 298, Z 73} c_vel
LIN {X 90, Y 291, Z 73} c_vel
LIN {X 99, Y 284, Z 73} c_vel
LIN {X 106, Y 277, Z 73} c_vel
LIN {X 113, Y 269, Z 73} c_vel
LIN {X 118, Y 261, Z 73} c_vel
LIN {X 123, Y 253, Z 73} c_vel
LIN {X 127, Y 244, Z 73} c_vel
LIN {X 130, Y 235, Z 73} c_vel
LIN {X 131, Y 226, Z 73} c_vel
LIN {X 133, Y 217, Z 73} c_vel
LIN {X 133, Y 207, Z 73} c_vel
LIN {X 133, Y 197, Z 73} c_vel
LIN {X 131, Y 186, Z 73} c_vel
LIN {X 129, Y 173, Z 73} c_vel
LIN {X 126, Y 160, Z 73} c_vel
LIN {X 120, Y 138, Z 73} c_vel
LIN {X 115, Y 118, Z 73} c_vel
LIN {X 112, Y 106, Z 73} c_vel
LIN {X 111, Y 96, Z 73} c_vel
LIN {X 110, Y 88, Z 73} c_vel
LIN {X 110, Y 81, Z 73} c_vel
LIN {X 111, Y 74, Z 73} c_vel
LIN {X 113, Y 69, Z 73} c_vel
LIN {X 116, Y 63, Z 73} c_vel
LIN {X 119, Y 58, Z 73} c_vel
LIN {X 124, Y 53, Z 73} c_vel
LIN {X 130, Y 48, Z 73} c_vel
LIN {X 138, Y 43, Z 73} c_vel
LIN {X 111, Y 0, Z 73} c_vel
$OUT[4] = FALSE
WAIT SEC 10.0
LIN {X 111, Y 0, Z 74} c_vel
$OUT[4] = TRUE
LIN {X 111, Y 0, Z 74} c_vel
LIN {X 106, Y 3, Z 74} c_vel
LIN {X 97, Y 9, Z 74} c_vel
LIN {X 89, Y 16, Z 74} c_vel
LIN {X 83, Y 23, Z 74} c_vel
LIN {X 77, Y 31, Z 74} c_vel
LIN {X 71, Y 39, Z 74} c_vel
LIN {X 67, Y 47, Z 74} c_vel
LIN {X 64, Y 56, Z 74} c_vel
LIN {X 62, Y 64, Z 74} c_vel
LIN {X 60, Y 73, Z 74} c_vel
LIN {X 59, Y 82, Z 74} c_vel
LIN {X 59, Y 92, Z 74} c_vel
LIN {X 59, Y 92, Z 74} c_vel
LIN {X 60, Y 103, Z 74} c_vel
LIN {X 62, Y 114, Z 74} c_vel
LIN {X 65, Y 127, Z 74} c_vel
LIN {X 69, Y 144, Z 74} c_vel
LIN {X 74, Y 163, Z 74} c_vel
LIN {X 79, Y 180, Z 74} c_vel
LIN {X 81, Y 191, Z 74} c_vel
LIN {X 82, Y 201, Z 74} c_vel
LIN {X 82, Y 209, Z 74} c_vel
LIN {X 82, Y 217, Z 74} c_vel
LIN {X 80, Y 223, Z 74} c_vel
LIN {X 78, Y 229, Z 74} c_vel
LIN {X 75, Y 234, Z 74} c_vel
LIN {X 71, Y 240, Z 74} c_vel
LIN {X 66, Y 245, Z 74} c_vel
LIN {X 60, Y 250, Z 74} c_vel
LIN {X 52, Y 256, Z 74} c_vel
LIN {X 42, Y 261, Z 74} c_vel
LIN {X 30, Y 267, Z 74} c_vel
LIN {X 16, Y 273, Z 74} c_vel
LIN {X 0, Y 278, Z 74} c_vel
LIN {X 14, Y 327, Z 74} c_vel
LIN {X 28, Y 322, Z 74} c_vel
LIN {X 43, Y 317, Z 74} c_vel
LIN {X 57, Y 311, Z 74} c_vel
LIN {X 70, Y 304, Z 74} c_vel
LIN {X 81, Y 298, Z 74} c_vel
LIN {X 90, Y 291, Z 74} c_vel
LIN {X 99, Y 284, Z 74} c_vel
LIN {X 106, Y 277, Z 74} c_vel
LIN {X 113, Y 269, Z 74} c_vel
LIN {X 118, Y 261, Z 74} c_vel
LIN {X 123, Y 253, Z 74} c_vel
LIN {X 127, Y 244, Z 74} c_vel
LIN {X 130, Y 235, Z 74} c_vel
LIN {X 131, Y 226, Z 74} c_vel
LIN {X 133, Y 217, Z 74} c_vel
LIN {X 133, Y 207, Z 74} c_vel
LIN {X 133, Y 197, Z 74} c_vel
LIN {X 131, Y 186, Z 74} c_vel
LIN {X 129, Y 173, Z 74} c_vel
LIN {X 126, Y 160, Z 74} c_vel
LIN {X 120, Y 138, Z 74} c_vel
LIN {X 115, Y 118, Z 74} c_vel
LIN {X 112, Y 106, Z 74} c_vel
LIN {X 111, Y 96, Z 74} c_vel
LIN {X 110, Y 88, Z 74} c_vel
LIN {X 110, Y 81, Z 74} c_vel
LIN {X 111, Y 74, Z 74} c_vel
LIN {X 113, Y 69, Z 74} c_vel
LIN {X 116, Y 63, Z 74} c_vel
LIN {X 119, Y 58, Z 74} c_vel
LIN {X 124, Y 53, Z 74} c_vel
LIN {X 130, Y 48, Z 74} c_vel
LIN {X 138, Y 43, Z 74} c_vel
LIN {X 111, Y 0, Z 74} c_vel
$OUT[4] = FALSE
WAIT SEC 10.0
LIN {X 111, Y 0, Z 75} c_vel
$OUT[4] = TRUE
LIN {X 111, Y 0, Z 75} c_vel
LIN {X 106, Y 3, Z 75} c_vel
LIN {X 97, Y 9, Z 75} c_vel
LIN {X 89, Y 16, Z 75} c_vel
LIN {X 83, Y 23, Z 75} c_vel
LIN {X 77, Y 31, Z 75} c_vel
LIN {X 71, Y 39, Z 75} c_vel
LIN {X 67, Y 47, Z 75} c_vel
LIN {X 64, Y 56, Z 75} c_vel
LIN {X 62, Y 64, Z 75} c_vel
LIN {X 60, Y 73, Z 75} c_vel
LIN {X 59, Y 82, Z 75} c_vel
LIN {X 59, Y 92, Z 75} c_vel
LIN {X 59, Y 92, Z 75} c_vel
LIN {X 60, Y 103, Z 75} c_vel
LIN {X 62, Y 114, Z 75} c_vel
LIN {X 65, Y 127, Z 75} c_vel
LIN {X 69, Y 144, Z 75} c_vel
LIN {X 74, Y 163, Z 75} c_vel
LIN {X 79, Y 180, Z 75} c_vel
LIN {X 81, Y 191, Z 75} c_vel
LIN {X 82, Y 201, Z 75} c_vel
LIN {X 82, Y 209, Z 75} c_vel
LIN {X 82, Y 217, Z 75} c_vel
LIN {X 80, Y 223, Z 75} c_vel
LIN {X 78, Y 229, Z 75} c_vel
LIN {X 75, Y 234, Z 75} c_vel
LIN {X 71, Y 240, Z 75} c_vel
LIN {X 66, Y 245, Z 75} c_vel
LIN {X 60, Y 250, Z 75} c_vel
LIN {X 52, Y 256, Z 75} c_vel
LIN {X 42, Y 261, Z 75} c_vel
LIN {X 30, Y 267, Z 75} c_vel
LIN {X 16, Y 273, Z 75} c_vel
LIN {X 0, Y 278, Z 75} c_vel
LIN {X 14, Y 327, Z 75} c_vel
LIN {X 28, Y 322, Z 75} c_vel
LIN {X 43, Y 317, Z 75} c_vel
LIN {X 57, Y 311, Z 75} c_vel
LIN {X 70, Y 304, Z 75} c_vel
LIN {X 81, Y 298, Z 75} c_vel
LIN {X 90, Y 291, Z 75} c_vel
LIN {X 99, Y 284, Z 75} c_vel
LIN {X 106, Y 277, Z 75} c_vel
LIN {X 113, Y 269, Z 75} c_vel
LIN {X 118, Y 261, Z 75} c_vel
LIN {X 123, Y 253, Z 75} c_vel
LIN {X 127, Y 244, Z 75} c_vel
LIN {X 130, Y 235, Z 75} c_vel
LIN {X 131, Y 226, Z 75} c_vel
LIN {X 133, Y 217, Z 75} c_vel
LIN {X 133, Y 207, Z 75} c_vel
LIN {X 133, Y 197, Z 75} c_vel
LIN {X 131, Y 186, Z 75} c_vel
LIN {X 129, Y 173, Z 75} c_vel
LIN {X 126, Y 160, Z 75} c_vel
LIN {X 120, Y 138, Z 75} c_vel
LIN {X 115, Y 118, Z 75} c_vel
LIN {X 112, Y 106, Z 75} c_vel
LIN {X 111, Y 96, Z 75} c_vel
LIN {X 110, Y 88, Z 75} c_vel
LIN {X 110, Y 81, Z 75} c_vel
LIN {X 111, Y 74, Z 75} c_vel
LIN {X 113, Y 69, Z 75} c_vel
LIN {X 116, Y 63, Z 75} c_vel
LIN {X 119, Y 58, Z 75} c_vel
LIN {X 124, Y 53, Z 75} c_vel
LIN {X 130, Y 48, Z 75} c_vel
LIN {X 138, Y 43, Z 75} c_vel
LIN {X 111, Y 0, Z 75} c_vel
$OUT[4] = FALSE
WAIT SEC 10.0
LIN {X 111, Y 0, Z 76} c_vel
$OUT[4] = TRUE
LIN {X 111, Y 0, Z 76} c_vel
LIN {X 106, Y 3, Z 76} c_vel
LIN {X 97, Y 9, Z 76} c_vel
LIN {X 89, Y 16, Z 76} c_vel
LIN {X 83, Y 23, Z 76} c_vel
LIN {X 77, Y 31, Z 76} c_vel
LIN {X 71, Y 39, Z 76} c_vel
LIN {X 67, Y 47, Z 76} c_vel
LIN {X 64, Y 56, Z 76} c_vel
LIN {X 62, Y 64, Z 76} c_vel
LIN {X 60, Y 73, Z 76} c_vel
LIN {X 59, Y 82, Z 76} c_vel
LIN {X 59, Y 92, Z 76} c_vel
LIN {X 59, Y 92, Z 76} c_vel
LIN {X 60, Y 103, Z 76} c_vel
LIN {X 62, Y 114, Z 76} c_vel
LIN {X 65, Y 127, Z 76} c_vel
LIN {X 69, Y 144, Z 76} c_vel
LIN {X 74, Y 163, Z 76} c_vel
LIN {X 79, Y 180, Z 76} c_vel
LIN {X 81, Y 191, Z 76} c_vel
LIN {X 82, Y 201, Z 76} c_vel
LIN {X 82, Y 209, Z 76} c_vel
LIN {X 82, Y 217, Z 76} c_vel
LIN {X 80, Y 223, Z 76} c_vel
LIN {X 78, Y 229, Z 76} c_vel
LIN {X 75, Y 234, Z 76} c_vel
LIN {X 71, Y 240, Z 76} c_vel
LIN {X 66, Y 245, Z 76} c_vel
LIN {X 60, Y 250, Z 76} c_vel
LIN {X 52, Y 256, Z 76} c_vel
LIN {X 42, Y 261, Z 76} c_vel
LIN {X 30, Y 267, Z 76} c_vel
LIN {X 16, Y 273, Z 76} c_vel
LIN {X 0, Y 278, Z 76} c_vel
LIN {X 14, Y 327, Z 76} c_vel
LIN {X 28, Y 322, Z 76} c_vel
LIN {X 43, Y 317, Z 76} c_vel
LIN {X 57, Y 311, Z 76} c_vel
LIN {X 70, Y 304, Z 76} c_vel
LIN {X 81, Y 298, Z 76} c_vel
LIN {X 90, Y 291, Z 76} c_vel
LIN {X 99, Y 284, Z 76} c_vel
LIN {X 106, Y 277, Z 76} c_vel
LIN {X 113, Y 269, Z 76} c_vel
LIN {X 118, Y 261, Z 76} c_vel
LIN {X 123, Y 253, Z 76} c_vel
LIN {X 127, Y 244, Z 76} c_vel
LIN {X 130, Y 235, Z 76} c_vel
LIN {X 131, Y 226, Z 76} c_vel
LIN {X 133, Y 217, Z 76} c_vel
LIN {X 133, Y 207, Z 76} c_vel
LIN {X 133, Y 197, Z 76} c_vel
LIN {X 131, Y 186, Z 76} c_vel
LIN {X 129, Y 173, Z 76} c_vel
LIN {X 126, Y 160, Z 76} c_vel
LIN {X 120, Y 138, Z 76} c_vel
LIN {X 115, Y 118, Z 76} c_vel
LIN {X 112, Y 106, Z 76} c_vel
LIN {X 111, Y 96, Z 76} c_vel
LIN {X 110, Y 88, Z 76} c_vel
LIN {X 110, Y 81, Z 76} c_vel
LIN {X 111, Y 74, Z 76} c_vel
LIN {X 113, Y 69, Z 76} c_vel
LIN {X 116, Y 63, Z 76} c_vel
LIN {X 119, Y 58, Z 76} c_vel
LIN {X 124, Y 53, Z 76} c_vel
LIN {X 130, Y 48, Z 76} c_vel
LIN {X 138, Y 43, Z 76} c_vel
LIN {X 111, Y 0, Z 76} c_vel
$OUT[4] = FALSE
WAIT SEC 10.0
END
